FUNCTION "MOTOR" : VOID	// FC 101
AUTHOR : gaw-be
FAMILY : MOTOR
NAME : MOTOR
VERSION : 0.1
BEGIN
// (block stored without names or comments; labels and parameter names are numbered)
NETWORK
TITLE =
      BLD   5;
      T     LD 103;
      TAK;
      T     LD 107;
      L     P##PARAM9;
      LAR1;
      L     W [AR1,P#0.0];
      T     LW 101;
      OPN   DB [LW 101];
      L     D [AR1,P#2.0];
      LAR1;
      L     LD 107;
      L     LD 103;
      L     W [AR1,P#2.0];
      L     -1;
      ==I;
      BLD   5;
      T     LD 103;
      TAK;
      T     LD 107;
      L     P##PARAM9;
      LAR1;
      L     W [AR1,P#0.0];
      T     LW 101;
      OPN   DB [LW 101];
      L     D [AR1,P#2.0];
      LAR1;
      L     LD 107;
      L     LD 103;
      R      [AR1,P#4.0];
      L     #PARAM5;
      BLD   5;
      T     LD 103;
      TAK;
      T     LD 107;
      L     P##PARAM9;
      LAR1;
      L     W [AR1,P#0.0];
      T     LW 101;
      OPN   DB [LW 101];
      L     D [AR1,P#2.0];
      LAR1;
      L     LD 107;
      L     LD 103;
      L     W [AR1,P#2.0];
      <>I;
      JC    M002;
      BLD   5;
      T     LD 103;
      TAK;
      T     LD 107;
      L     P##PARAM9;
      LAR1;
      L     W [AR1,P#0.0];
      T     LW 101;
      OPN   DB [LW 101];
      L     D [AR1,P#2.0];
      LAR1;
      L     LD 107;
      L     LD 103;
      A      [AR1,P#4.0];
      JC    M001;
      BLD   5;
      T     LD 103;
      TAK;
      T     LD 107;
      L     P##PARAM8;
      LAR1;
      L     W [AR1,P#0.0];
      T     LW 101;
      OPN   DB [LW 101];
      L     D [AR1,P#2.0];
      LAR1;
      L     LD 107;
      L     LD 103;
      A      [AR1,P#0.0];
      BLD   5;
      T     LD 103;
      TAK;
      T     LD 107;
      L     P##PARAM9;
      LAR1;
      L     W [AR1,P#0.0];
      T     LW 101;
      OPN   DB [LW 101];
      L     D [AR1,P#2.0];
      LAR1;
      L     LD 107;
      L     LD 103;
      =      [AR1,P#0.0];
      BLD   5;
      T     LD 103;
      TAK;
      T     LD 107;
      L     P##PARAM8;
      LAR1;
      L     W [AR1,P#0.0];
      T     LW 101;
      OPN   DB [LW 101];
      L     D [AR1,P#2.0];
      LAR1;
      L     LD 107;
      L     LD 103;
      A      [AR1,P#0.1];
      BLD   5;
      T     LD 103;
      TAK;
      T     LD 107;
      L     P##PARAM9;
      LAR1;
      L     W [AR1,P#0.0];
      T     LW 101;
      OPN   DB [LW 101];
      L     D [AR1,P#2.0];
      LAR1;
      L     LD 107;
      L     LD 103;
      =      [AR1,P#0.1];
      BLD   5;
      T     LD 103;
      TAK;
      T     LD 107;
      L     P##PARAM8;
      LAR1;
      L     W [AR1,P#0.0];
      T     LW 101;
      OPN   DB [LW 101];
      L     D [AR1,P#2.0];
      LAR1;
      L     LD 107;
      L     LD 103;
      A      [AR1,P#0.3];
      BLD   5;
      T     LD 103;
      TAK;
      T     LD 107;
      L     P##PARAM9;
      LAR1;
      L     W [AR1,P#0.0];
      T     LW 101;
      OPN   DB [LW 101];
      L     D [AR1,P#2.0];
      LAR1;
      L     LD 107;
      L     LD 103;
      =      [AR1,P#0.3];
      SET;
      BLD   5;
      T     LD 103;
      TAK;
      T     LD 107;
      L     P##PARAM9;
      LAR1;
      L     W [AR1,P#0.0];
      T     LW 101;
      OPN   DB [LW 101];
      L     D [AR1,P#2.0];
      LAR1;
      L     LD 107;
      L     LD 103;
      =      [AR1,P#4.0];
M001: BLD   5;
      T     LD 103;
      TAK;
      T     LD 107;
      L     P##PARAM9;
      LAR1;
      L     W [AR1,P#0.0];
      T     LW 101;
      OPN   DB [LW 101];
      L     D [AR1,P#2.0];
      LAR1;
      L     LD 107;
      L     LD 103;
      A      [AR1,P#0.0];
      BLD   5;
      T     LD 103;
      TAK;
      T     LD 107;
      L     P##PARAM8;
      LAR1;
      L     W [AR1,P#0.0];
      T     LW 101;
      OPN   DB [LW 101];
      L     D [AR1,P#2.0];
      LAR1;
      L     LD 107;
      L     LD 103;
      =      [AR1,P#0.0];
      BLD   5;
      T     LD 103;
      TAK;
      T     LD 107;
      L     P##PARAM9;
      LAR1;
      L     W [AR1,P#0.0];
      T     LW 101;
      OPN   DB [LW 101];
      L     D [AR1,P#2.0];
      LAR1;
      L     LD 107;
      L     LD 103;
      A      [AR1,P#0.1];
      BLD   5;
      T     LD 103;
      TAK;
      T     LD 107;
      L     P##PARAM8;
      LAR1;
      L     W [AR1,P#0.0];
      T     LW 101;
      OPN   DB [LW 101];
      L     D [AR1,P#2.0];
      LAR1;
      L     LD 107;
      L     LD 103;
      =      [AR1,P#0.1];
      BLD   5;
      T     LD 103;
      TAK;
      T     LD 107;
      L     P##PARAM8;
      LAR1;
      L     W [AR1,P#0.0];
      T     LW 101;
      OPN   DB [LW 101];
      L     D [AR1,P#2.0];
      LAR1;
      L     LD 107;
      L     LD 103;
      A      [AR1,P#0.2];
      BLD   5;
      T     LD 103;
      TAK;
      T     LD 107;
      L     P##PARAM9;
      LAR1;
      L     W [AR1,P#0.0];
      T     LW 101;
      OPN   DB [LW 101];
      L     D [AR1,P#2.0];
      LAR1;
      L     LD 107;
      L     LD 103;
      =      [AR1,P#0.2];
      BLD   5;
      T     LD 103;
      TAK;
      T     LD 107;
      L     P##PARAM9;
      LAR1;
      L     W [AR1,P#0.0];
      T     LW 101;
      OPN   DB [LW 101];
      L     D [AR1,P#2.0];
      LAR1;
      L     LD 107;
      L     LD 103;
      A      [AR1,P#0.3];
      BLD   5;
      T     LD 103;
      TAK;
      T     LD 107;
      L     P##PARAM8;
      LAR1;
      L     W [AR1,P#0.0];
      T     LW 101;
      OPN   DB [LW 101];
      L     D [AR1,P#2.0];
      LAR1;
      L     LD 107;
      L     LD 103;
      =      [AR1,P#0.3];
      BLD   5;
      T     LD 103;
      TAK;
      T     LD 107;
      L     P##PARAM8;
      LAR1;
      L     W [AR1,P#0.0];
      T     LW 101;
      OPN   DB [LW 101];
      L     D [AR1,P#2.0];
      LAR1;
      L     LD 107;
      L     LD 103;
      A      [AR1,P#0.4];
      BLD   5;
      T     LD 103;
      TAK;
      T     LD 107;
      L     P##PARAM9;
      LAR1;
      L     W [AR1,P#0.0];
      T     LW 101;
      OPN   DB [LW 101];
      L     D [AR1,P#2.0];
      LAR1;
      L     LD 107;
      L     LD 103;
      =      [AR1,P#0.4];
      BLD   5;
      T     LD 103;
      TAK;
      T     LD 107;
      L     P##PARAM8;
      LAR1;
      L     W [AR1,P#0.0];
      T     LW 101;
      OPN   DB [LW 101];
      L     D [AR1,P#2.0];
      LAR1;
      L     LD 107;
      L     LD 103;
      A      [AR1,P#0.5];
      BLD   5;
      T     LD 103;
      TAK;
      T     LD 107;
      L     P##PARAM9;
      LAR1;
      L     W [AR1,P#0.0];
      T     LW 101;
      OPN   DB [LW 101];
      L     D [AR1,P#2.0];
      LAR1;
      L     LD 107;
      L     LD 103;
      =      [AR1,P#0.5];
      BLD   5;
      T     LD 103;
      TAK;
      T     LD 107;
      L     P##PARAM8;
      LAR1;
      L     W [AR1,P#0.0];
      T     LW 101;
      OPN   DB [LW 101];
      L     D [AR1,P#2.0];
      LAR1;
      L     LD 107;
      L     LD 103;
      A      [AR1,P#0.6];
      BLD   5;
      T     LD 103;
      TAK;
      T     LD 107;
      L     P##PARAM9;
      LAR1;
      L     W [AR1,P#0.0];
      T     LW 101;
      OPN   DB [LW 101];
      L     D [AR1,P#2.0];
      LAR1;
      L     LD 107;
      L     LD 103;
      =      [AR1,P#0.6];
      BLD   5;
      T     LD 103;
      TAK;
      T     LD 107;
      L     P##PARAM8;
      LAR1;
      L     W [AR1,P#0.0];
      T     LW 101;
      OPN   DB [LW 101];
      L     D [AR1,P#2.0];
      LAR1;
      L     LD 107;
      L     LD 103;
      A      [AR1,P#0.7];
      BLD   5;
      T     LD 103;
      TAK;
      T     LD 107;
      L     P##PARAM9;
      LAR1;
      L     W [AR1,P#0.0];
      T     LW 101;
      OPN   DB [LW 101];
      L     D [AR1,P#2.0];
      LAR1;
      L     LD 107;
      L     LD 103;
      =      [AR1,P#0.7];
      BLD   5;
      T     LD 103;
      TAK;
      T     LD 107;
      L     P##PARAM8;
      LAR1;
      L     W [AR1,P#0.0];
      T     LW 101;
      OPN   DB [LW 101];
      L     D [AR1,P#2.0];
      LAR1;
      L     LD 107;
      L     LD 103;
      L     B [AR1,P#1.0];
      BLD   5;
      T     LD 103;
      TAK;
      T     LD 107;
      L     P##PARAM9;
      LAR1;
      L     W [AR1,P#0.0];
      T     LW 101;
      OPN   DB [LW 101];
      L     D [AR1,P#2.0];
      LAR1;
      L     LD 107;
      L     LD 103;
      T     B [AR1,P#1.0];
M002: NOP   0;
NETWORK
TITLE =
      A(;
      A     #PARAM3;
      BLD   5;
      T     LD 103;
      TAK;
      T     LD 107;
      L     P##PARAM8;
      LAR1;
      L     W [AR1,P#0.0];
      T     LW 101;
      OPN   DB [LW 101];
      L     D [AR1,P#2.0];
      LAR1;
      L     LD 107;
      L     LD 103;
      AN     [AR1,P#0.0];
      O;
      BLD   5;
      T     LD 103;
      TAK;
      T     LD 107;
      L     P##PARAM8;
      LAR1;
      L     W [AR1,P#0.0];
      T     LW 101;
      OPN   DB [LW 101];
      L     D [AR1,P#2.0];
      LAR1;
      L     LD 107;
      L     LD 103;
      A      [AR1,P#0.0];
      BLD   5;
      T     LD 103;
      TAK;
      T     LD 107;
      L     P##PARAM8;
      LAR1;
      L     W [AR1,P#0.0];
      T     LW 101;
      OPN   DB [LW 101];
      L     D [AR1,P#2.0];
      LAR1;
      L     LD 107;
      L     LD 103;
      A      [AR1,P#0.1];
      );
      AN    #PARAM4;
      AN    #PARAM2;
      =     L 0.0;
      =     #PARAM6;
NETWORK
TITLE =
      A     #PARAM2;
      BLD   5;
      T     LD 103;
      TAK;
      T     LD 107;
      L     P##PARAM8;
      LAR1;
      L     W [AR1,P#0.0];
      T     LW 101;
      OPN   DB [LW 101];
      L     D [AR1,P#2.0];
      LAR1;
      L     LD 107;
      L     LD 103;
      =      [AR1,P#0.2];
NETWORK
TITLE =
      BLD   5;
      T     LD 103;
      TAK;
      T     LD 107;
      L     P##PARAM8;
      LAR1;
      L     W [AR1,P#0.0];
      T     LW 101;
      OPN   DB [LW 101];
      L     D [AR1,P#2.0];
      LAR1;
      L     LD 107;
      L     LD 103;
      A      [AR1,P#0.2];
      BLD   5;
      T     LD 103;
      TAK;
      T     LD 107;
      L     P##PARAM8;
      LAR1;
      L     W [AR1,P#0.0];
      T     LW 101;
      OPN   DB [LW 101];
      L     D [AR1,P#2.0];
      LAR1;
      L     LD 107;
      L     LD 103;
      A      [AR1,P#0.3];
      BLD   5;
      T     LD 103;
      TAK;
      T     LD 107;
      L     P##PARAM8;
      LAR1;
      L     W [AR1,P#0.0];
      T     LW 101;
      OPN   DB [LW 101];
      L     D [AR1,P#2.0];
      LAR1;
      L     LD 107;
      L     LD 103;
      R      [AR1,P#0.2];
NETWORK
TITLE =
      A     L 0.0;
      AN    #PARAM1;
      O;
      AN    L 0.0;
      A     #PARAM1;
      BLD   5;
      T     LD 103;
      TAK;
      T     LD 107;
      L     P##PARAM8;
      LAR1;
      L     W [AR1,P#0.0];
      T     LW 101;
      OPN   DB [LW 101];
      L     D [AR1,P#2.0];
      LAR1;
      L     LD 107;
      L     LD 103;
      O      [AR1,P#0.2];
      =     #PARAM7;
NETWORK
TITLE =
      AN    #PARAM1;
      AN    #PARAM2;
      BLD   5;
      T     LD 103;
      TAK;
      T     LD 107;
      L     P##PARAM8;
      LAR1;
      L     W [AR1,P#0.0];
      T     LW 101;
      OPN   DB [LW 101];
      L     D [AR1,P#2.0];
      LAR1;
      L     LD 107;
      L     LD 103;
      =      [AR1,P#0.4];
NETWORK
TITLE =
      A     #PARAM1;
      AN    #PARAM2;
      BLD   5;
      T     LD 103;
      TAK;
      T     LD 107;
      L     P##PARAM8;
      LAR1;
      L     W [AR1,P#0.0];
      T     LW 101;
      OPN   DB [LW 101];
      L     D [AR1,P#2.0];
      LAR1;
      L     LD 107;
      L     LD 103;
      =      [AR1,P#0.5];
NETWORK
TITLE =
      A     #PARAM2;
      A     M 0.7;
      BLD   5;
      T     LD 103;
      TAK;
      T     LD 107;
      L     P##PARAM8;
      LAR1;
      L     W [AR1,P#0.0];
      T     LW 101;
      OPN   DB [LW 101];
      L     D [AR1,P#2.0];
      LAR1;
      L     LD 107;
      L     LD 103;
      =      [AR1,P#0.6];
NETWORK
TITLE =
      A     #PARAM2;
      AN    M 0.7;
      BLD   5;
      T     LD 103;
      TAK;
      T     LD 107;
      L     P##PARAM8;
      LAR1;
      L     W [AR1,P#0.0];
      T     LW 101;
      OPN   DB [LW 101];
      L     D [AR1,P#2.0];
      LAR1;
      L     LD 107;
      L     LD 103;
      =      [AR1,P#0.7];
NETWORK
TITLE =
      BLD   5;
      T     LD 103;
      TAK;
      T     LD 107;
      L     P##PARAM8;
      LAR1;
      L     W [AR1,P#0.0];
      T     LW 101;
      OPN   DB [LW 101];
      L     D [AR1,P#2.0];
      LAR1;
      L     LD 107;
      L     LD 103;
      A      [AR1,P#0.3];
      BLD   5;
      T     LD 103;
      TAK;
      T     LD 107;
      L     P##PARAM8;
      LAR1;
      L     W [AR1,P#0.0];
      T     LW 101;
      OPN   DB [LW 101];
      L     D [AR1,P#2.0];
      LAR1;
      L     LD 107;
      L     LD 103;
      R      [AR1,P#0.3];
NETWORK
TITLE =
      BLD   5;
      T     LD 103;
      TAK;
      T     LD 107;
      L     P##PARAM8;
      LAR1;
      L     W [AR1,P#0.0];
      T     LW 101;
      OPN   DB [LW 101];
      L     D [AR1,P#2.0];
      LAR1;
      L     LD 107;
      L     LD 103;
      A      [AR1,P#0.0];
      =     L 100.0;
      BLD   5;
      T     LD 103;
      TAK;
      T     LD 107;
      L     P##PARAM8;
      LAR1;
      L     W [AR1,P#0.0];
      T     LW 101;
      OPN   DB [LW 101];
      L     D [AR1,P#2.0];
      LAR1;
      L     LD 107;
      L     LD 103;
      A      [AR1,P#0.1];
      =     L 100.1;
      BLD   5;
      T     LD 103;
      TAK;
      T     LD 107;
      L     P##PARAM8;
      LAR1;
      L     W [AR1,P#0.0];
      T     LW 101;
      OPN   DB [LW 101];
      L     D [AR1,P#2.0];
      LAR1;
      L     LD 107;
      L     LD 103;
      A      [AR1,P#0.2];
      =     L 100.2;
      BLD   5;
      T     LD 103;
      TAK;
      T     LD 107;
      L     P##PARAM8;
      LAR1;
      L     W [AR1,P#0.0];
      T     LW 101;
      OPN   DB [LW 101];
      L     D [AR1,P#2.0];
      LAR1;
      L     LD 107;
      L     LD 103;
      A      [AR1,P#0.3];
      =     L 100.3;
      BLD   5;
      T     LD 103;
      TAK;
      T     LD 107;
      L     P##PARAM8;
      LAR1;
      L     W [AR1,P#0.0];
      T     LW 101;
      OPN   DB [LW 101];
      L     D [AR1,P#2.0];
      LAR1;
      L     LD 107;
      L     LD 103;
      A      [AR1,P#0.4];
      =     L 100.4;
      BLD   5;
      T     LD 103;
      TAK;
      T     LD 107;
      L     P##PARAM8;
      LAR1;
      L     W [AR1,P#0.0];
      T     LW 101;
      OPN   DB [LW 101];
      L     D [AR1,P#2.0];
      LAR1;
      L     LD 107;
      L     LD 103;
      A      [AR1,P#0.5];
      =     L 100.5;
      BLD   5;
      T     LD 103;
      TAK;
      T     LD 107;
      L     P##PARAM8;
      LAR1;
      L     W [AR1,P#0.0];
      T     LW 101;
      OPN   DB [LW 101];
      L     D [AR1,P#2.0];
      LAR1;
      L     LD 107;
      L     LD 103;
      A      [AR1,P#0.6];
      =     L 100.6;
      BLD   5;
      T     LD 103;
      TAK;
      T     LD 107;
      L     P##PARAM8;
      LAR1;
      L     W [AR1,P#0.0];
      T     LW 101;
      OPN   DB [LW 101];
      L     D [AR1,P#2.0];
      LAR1;
      L     LD 107;
      L     LD 103;
      A      [AR1,P#0.7];
      =     L 100.7;
      L     LB 100;
      BLD   5;
      T     LD 103;
      TAK;
      T     LD 107;
      L     P##PARAM8;
      LAR1;
      L     W [AR1,P#0.0];
      T     LW 101;
      OPN   DB [LW 101];
      L     D [AR1,P#2.0];
      LAR1;
      L     LD 107;
      L     LD 103;
      T     B [AR1,P#1.0];
END_FUNCTION

FUNCTION "level" : VOID	// FC 107
AUTHOR : gaw-be
FAMILY : level
NAME : display
VERSION : 0.2
BEGIN
// (block stored without names or comments; labels and parameter names are numbered)
NETWORK
TITLE =
      L     #PARAM3;
      BLD   5;
      T     LD 106;
      TAK;
      T     LD 110;
      L     P##PARAM12;
      LAR1;
      L     W [AR1,P#0.0];
      T     LW 104;
      OPN   DB [LW 104];
      L     D [AR1,P#2.0];
      LAR1;
      L     LD 110;
      L     LD 106;
      T     B [AR1,P#28.0];
      BLD   5;
      T     LD 106;
      TAK;
      T     LD 110;
      L     P##PARAM13;
      LAR1;
      L     W [AR1,P#0.0];
      T     LW 104;
      OPN   DB [LW 104];
      L     D [AR1,P#2.0];
      LAR1;
      L     LD 110;
      L     LD 106;
      L     W [AR1,P#28.0];
      L     -1;
      ==I;
      BLD   5;
      T     LD 106;
      TAK;
      T     LD 110;
      L     P##PARAM13;
      LAR1;
      L     W [AR1,P#0.0];
      T     LW 104;
      OPN   DB [LW 104];
      L     D [AR1,P#2.0];
      LAR1;
      L     LD 110;
      L     LD 106;
      R      [AR1,P#30.0];
      L     #PARAM2;
      BLD   5;
      T     LD 106;
      TAK;
      T     LD 110;
      L     P##PARAM13;
      LAR1;
      L     W [AR1,P#0.0];
      T     LW 104;
      OPN   DB [LW 104];
      L     D [AR1,P#2.0];
      LAR1;
      L     LD 110;
      L     LD 106;
      L     W [AR1,P#28.0];
      <>I;
      JC    M010;
      BLD   5;
      T     LD 106;
      TAK;
      T     LD 110;
      L     P##PARAM13;
      LAR1;
      L     W [AR1,P#0.0];
      T     LW 104;
      OPN   DB [LW 104];
      L     D [AR1,P#2.0];
      LAR1;
      L     LD 110;
      L     LD 106;
      A      [AR1,P#30.0];
      JC    M001;
      BLD   5;
      T     LD 106;
      TAK;
      T     LD 110;
      L     P##PARAM12;
      LAR1;
      L     W [AR1,P#0.0];
      T     LW 104;
      OPN   DB [LW 104];
      L     D [AR1,P#2.0];
      LAR1;
      L     LD 110;
      L     LD 106;
      L     B [AR1,P#4.0];
      BLD   5;
      T     LD 106;
      TAK;
      T     LD 110;
      L     P##PARAM13;
      LAR1;
      L     W [AR1,P#0.0];
      T     LW 104;
      OPN   DB [LW 104];
      L     D [AR1,P#2.0];
      LAR1;
      L     LD 110;
      L     LD 106;
      T     B [AR1,P#4.0];
      BLD   5;
      T     LD 106;
      TAK;
      T     LD 110;
      L     P##PARAM12;
      LAR1;
      L     W [AR1,P#0.0];
      T     LW 104;
      OPN   DB [LW 104];
      L     D [AR1,P#2.0];
      LAR1;
      L     LD 110;
      L     LD 106;
      L     D [AR1,P#6.0];
      BLD   5;
      T     LD 106;
      TAK;
      T     LD 110;
      L     P##PARAM13;
      LAR1;
      L     W [AR1,P#0.0];
      T     LW 104;
      OPN   DB [LW 104];
      L     D [AR1,P#2.0];
      LAR1;
      L     LD 110;
      L     LD 106;
      T     D [AR1,P#6.0];
      BLD   5;
      T     LD 106;
      TAK;
      T     LD 110;
      L     P##PARAM12;
      LAR1;
      L     W [AR1,P#0.0];
      T     LW 104;
      OPN   DB [LW 104];
      L     D [AR1,P#2.0];
      LAR1;
      L     LD 110;
      L     LD 106;
      L     D [AR1,P#10.0];
      BLD   5;
      T     LD 106;
      TAK;
      T     LD 110;
      L     P##PARAM13;
      LAR1;
      L     W [AR1,P#0.0];
      T     LW 104;
      OPN   DB [LW 104];
      L     D [AR1,P#2.0];
      LAR1;
      L     LD 110;
      L     LD 106;
      T     D [AR1,P#10.0];
      BLD   5;
      T     LD 106;
      TAK;
      T     LD 110;
      L     P##PARAM12;
      LAR1;
      L     W [AR1,P#0.0];
      T     LW 104;
      OPN   DB [LW 104];
      L     D [AR1,P#2.0];
      LAR1;
      L     LD 110;
      L     LD 106;
      L     D [AR1,P#14.0];
      BLD   5;
      T     LD 106;
      TAK;
      T     LD 110;
      L     P##PARAM13;
      LAR1;
      L     W [AR1,P#0.0];
      T     LW 104;
      OPN   DB [LW 104];
      L     D [AR1,P#2.0];
      LAR1;
      L     LD 110;
      L     LD 106;
      T     D [AR1,P#14.0];
      BLD   5;
      T     LD 106;
      TAK;
      T     LD 110;
      L     P##PARAM12;
      LAR1;
      L     W [AR1,P#0.0];
      T     LW 104;
      OPN   DB [LW 104];
      L     D [AR1,P#2.0];
      LAR1;
      L     LD 110;
      L     LD 106;
      L     W [AR1,P#18.0];
      BLD   5;
      T     LD 106;
      TAK;
      T     LD 110;
      L     P##PARAM13;
      LAR1;
      L     W [AR1,P#0.0];
      T     LW 104;
      OPN   DB [LW 104];
      L     D [AR1,P#2.0];
      LAR1;
      L     LD 110;
      L     LD 106;
      T     W [AR1,P#18.0];
      BLD   5;
      T     LD 106;
      TAK;
      T     LD 110;
      L     P##PARAM12;
      LAR1;
      L     W [AR1,P#0.0];
      T     LW 104;
      OPN   DB [LW 104];
      L     D [AR1,P#2.0];
      LAR1;
      L     LD 110;
      L     LD 106;
      L     W [AR1,P#20.0];
      BLD   5;
      T     LD 106;
      TAK;
      T     LD 110;
      L     P##PARAM13;
      LAR1;
      L     W [AR1,P#0.0];
      T     LW 104;
      OPN   DB [LW 104];
      L     D [AR1,P#2.0];
      LAR1;
      L     LD 110;
      L     LD 106;
      T     W [AR1,P#20.0];
      BLD   5;
      T     LD 106;
      TAK;
      T     LD 110;
      L     P##PARAM12;
      LAR1;
      L     W [AR1,P#0.0];
      T     LW 104;
      OPN   DB [LW 104];
      L     D [AR1,P#2.0];
      LAR1;
      L     LD 110;
      L     LD 106;
      L     W [AR1,P#22.0];
      BLD   5;
      T     LD 106;
      TAK;
      T     LD 110;
      L     P##PARAM13;
      LAR1;
      L     W [AR1,P#0.0];
      T     LW 104;
      OPN   DB [LW 104];
      L     D [AR1,P#2.0];
      LAR1;
      L     LD 110;
      L     LD 106;
      T     W [AR1,P#22.0];
      BLD   5;
      T     LD 106;
      TAK;
      T     LD 110;
      L     P##PARAM12;
      LAR1;
      L     W [AR1,P#0.0];
      T     LW 104;
      OPN   DB [LW 104];
      L     D [AR1,P#2.0];
      LAR1;
      L     LD 110;
      L     LD 106;
      L     W [AR1,P#24.0];
      BLD   5;
      T     LD 106;
      TAK;
      T     LD 110;
      L     P##PARAM13;
      LAR1;
      L     W [AR1,P#0.0];
      T     LW 104;
      OPN   DB [LW 104];
      L     D [AR1,P#2.0];
      LAR1;
      L     LD 110;
      L     LD 106;
      T     W [AR1,P#24.0];
      BLD   5;
      T     LD 106;
      TAK;
      T     LD 110;
      L     P##PARAM12;
      LAR1;
      L     W [AR1,P#0.0];
      T     LW 104;
      OPN   DB [LW 104];
      L     D [AR1,P#2.0];
      LAR1;
      L     LD 110;
      L     LD 106;
      L     W [AR1,P#26.0];
      BLD   5;
      T     LD 106;
      TAK;
      T     LD 110;
      L     P##PARAM13;
      LAR1;
      L     W [AR1,P#0.0];
      T     LW 104;
      OPN   DB [LW 104];
      L     D [AR1,P#2.0];
      LAR1;
      L     LD 110;
      L     LD 106;
      T     W [AR1,P#26.0];
      BLD   5;
      T     LD 106;
      TAK;
      T     LD 110;
      L     P##PARAM12;
      LAR1;
      L     W [AR1,P#0.0];
      T     LW 104;
      OPN   DB [LW 104];
      L     D [AR1,P#2.0];
      LAR1;
      L     LD 110;
      L     LD 106;
      L     B [AR1,P#28.0];
      BLD   5;
      T     LD 106;
      TAK;
      T     LD 110;
      L     P##PARAM13;
      LAR1;
      L     W [AR1,P#0.0];
      T     LW 104;
      OPN   DB [LW 104];
      L     D [AR1,P#2.0];
      LAR1;
      L     LD 110;
      L     LD 106;
      T     B [AR1,P#31.0];
      BLD   5;
      T     LD 106;
      TAK;
      T     LD 110;
      L     P##PARAM12;
      LAR1;
      L     W [AR1,P#0.0];
      T     LW 104;
      OPN   DB [LW 104];
      L     D [AR1,P#2.0];
      LAR1;
      L     LD 110;
      L     LD 106;
      L     W [AR1,P#30.0];
      BLD   5;
      T     LD 106;
      TAK;
      T     LD 110;
      L     P##PARAM13;
      LAR1;
      L     W [AR1,P#0.0];
      T     LW 104;
      OPN   DB [LW 104];
      L     D [AR1,P#2.0];
      LAR1;
      L     LD 110;
      L     LD 106;
      T     W [AR1,P#32.0];
      BLD   5;
      T     LD 106;
      TAK;
      T     LD 110;
      L     P##PARAM12;
      LAR1;
      L     W [AR1,P#0.0];
      T     LW 104;
      OPN   DB [LW 104];
      L     D [AR1,P#2.0];
      LAR1;
      L     LD 110;
      L     LD 106;
      L     W [AR1,P#32.0];
      BLD   5;
      T     LD 106;
      TAK;
      T     LD 110;
      L     P##PARAM13;
      LAR1;
      L     W [AR1,P#0.0];
      T     LW 104;
      OPN   DB [LW 104];
      L     D [AR1,P#2.0];
      LAR1;
      L     LD 110;
      L     LD 106;
      T     W [AR1,P#34.0];
      BLD   5;
      T     LD 106;
      TAK;
      T     LD 110;
      L     P##PARAM12;
      LAR1;
      L     W [AR1,P#0.0];
      T     LW 104;
      OPN   DB [LW 104];
      L     D [AR1,P#2.0];
      LAR1;
      L     LD 110;
      L     LD 106;
      L     W [AR1,P#34.0];
      BLD   5;
      T     LD 106;
      TAK;
      T     LD 110;
      L     P##PARAM13;
      LAR1;
      L     W [AR1,P#0.0];
      T     LW 104;
      OPN   DB [LW 104];
      L     D [AR1,P#2.0];
      LAR1;
      L     LD 110;
      L     LD 106;
      T     W [AR1,P#36.0];
      BLD   5;
      T     LD 106;
      TAK;
      T     LD 110;
      L     P##PARAM12;
      LAR1;
      L     W [AR1,P#0.0];
      T     LW 104;
      OPN   DB [LW 104];
      L     D [AR1,P#2.0];
      LAR1;
      L     LD 110;
      L     LD 106;
      L     W [AR1,P#36.0];
      BLD   5;
      T     LD 106;
      TAK;
      T     LD 110;
      L     P##PARAM13;
      LAR1;
      L     W [AR1,P#0.0];
      T     LW 104;
      OPN   DB [LW 104];
      L     D [AR1,P#2.0];
      LAR1;
      L     LD 110;
      L     LD 106;
      T     W [AR1,P#38.0];
      BLD   5;
      T     LD 106;
      TAK;
      T     LD 110;
      L     P##PARAM12;
      LAR1;
      L     W [AR1,P#0.0];
      T     LW 104;
      OPN   DB [LW 104];
      L     D [AR1,P#2.0];
      LAR1;
      L     LD 110;
      L     LD 106;
      L     W [AR1,P#38.0];
      BLD   5;
      T     LD 106;
      TAK;
      T     LD 110;
      L     P##PARAM13;
      LAR1;
      L     W [AR1,P#0.0];
      T     LW 104;
      OPN   DB [LW 104];
      L     D [AR1,P#2.0];
      LAR1;
      L     LD 110;
      L     LD 106;
      T     W [AR1,P#40.0];
      BLD   5;
      T     LD 106;
      TAK;
      T     LD 110;
      L     P##PARAM12;
      LAR1;
      L     W [AR1,P#0.0];
      T     LW 104;
      OPN   DB [LW 104];
      L     D [AR1,P#2.0];
      LAR1;
      L     LD 110;
      L     LD 106;
      L     W [AR1,P#40.0];
      BLD   5;
      T     LD 106;
      TAK;
      T     LD 110;
      L     P##PARAM13;
      LAR1;
      L     W [AR1,P#0.0];
      T     LW 104;
      OPN   DB [LW 104];
      L     D [AR1,P#2.0];
      LAR1;
      L     LD 110;
      L     LD 106;
      T     W [AR1,P#42.0];
      BLD   5;
      T     LD 106;
      TAK;
      T     LD 110;
      L     P##PARAM12;
      LAR1;
      L     W [AR1,P#0.0];
      T     LW 104;
      OPN   DB [LW 104];
      L     D [AR1,P#2.0];
      LAR1;
      L     LD 110;
      L     LD 106;
      L     W [AR1,P#42.0];
      BLD   5;
      T     LD 106;
      TAK;
      T     LD 110;
      L     P##PARAM13;
      LAR1;
      L     W [AR1,P#0.0];
      T     LW 104;
      OPN   DB [LW 104];
      L     D [AR1,P#2.0];
      LAR1;
      L     LD 110;
      L     LD 106;
      T     W [AR1,P#44.0];
      BLD   5;
      T     LD 106;
      TAK;
      T     LD 110;
      L     P##PARAM12;
      LAR1;
      L     W [AR1,P#0.0];
      T     LW 104;
      OPN   DB [LW 104];
      L     D [AR1,P#2.0];
      LAR1;
      L     LD 110;
      L     LD 106;
      L     W [AR1,P#44.0];
      BLD   5;
      T     LD 106;
      TAK;
      T     LD 110;
      L     P##PARAM13;
      LAR1;
      L     W [AR1,P#0.0];
      T     LW 104;
      OPN   DB [LW 104];
      L     D [AR1,P#2.0];
      LAR1;
      L     LD 110;
      L     LD 106;
      T     W [AR1,P#46.0];
      SET;
      BLD   5;
      T     LD 106;
      TAK;
      T     LD 110;
      L     P##PARAM13;
      LAR1;
      L     W [AR1,P#0.0];
      T     LW 104;
      OPN   DB [LW 104];
      L     D [AR1,P#2.0];
      LAR1;
      L     LD 110;
      L     LD 106;
      =      [AR1,P#30.0];
M001: BLD   5;
      T     LD 106;
      TAK;
      T     LD 110;
      L     P##PARAM12;
      LAR1;
      L     W [AR1,P#0.0];
      T     LW 104;
      OPN   DB [LW 104];
      L     D [AR1,P#2.0];
      LAR1;
      L     LD 110;
      L     LD 106;
      L     D [AR1,P#0.0];
      BLD   5;
      T     LD 106;
      TAK;
      T     LD 110;
      L     P##PARAM13;
      LAR1;
      L     W [AR1,P#0.0];
      T     LW 104;
      OPN   DB [LW 104];
      L     D [AR1,P#2.0];
      LAR1;
      L     LD 110;
      L     LD 106;
      T     D [AR1,P#0.0];
      BLD   5;
      T     LD 106;
      TAK;
      T     LD 110;
      L     P##PARAM13;
      LAR1;
      L     W [AR1,P#0.0];
      T     LW 104;
      OPN   DB [LW 104];
      L     D [AR1,P#2.0];
      LAR1;
      L     LD 110;
      L     LD 106;
      L     B [AR1,P#4.0];
      BLD   5;
      T     LD 106;
      TAK;
      T     LD 110;
      L     P##PARAM12;
      LAR1;
      L     W [AR1,P#0.0];
      T     LW 104;
      OPN   DB [LW 104];
      L     D [AR1,P#2.0];
      LAR1;
      L     LD 110;
      L     LD 106;
      T     B [AR1,P#4.0];
      BLD   5;
      T     LD 106;
      TAK;
      T     LD 110;
      L     P##PARAM13;
      LAR1;
      L     W [AR1,P#0.0];
      T     LW 104;
      OPN   DB [LW 104];
      L     D [AR1,P#2.0];
      LAR1;
      L     LD 110;
      L     LD 106;
      L     D [AR1,P#10.0];
      BLD   5;
      T     LD 106;
      TAK;
      T     LD 110;
      L     P##PARAM12;
      LAR1;
      L     W [AR1,P#0.0];
      T     LW 104;
      OPN   DB [LW 104];
      L     D [AR1,P#2.0];
      LAR1;
      L     LD 110;
      L     LD 106;
      T     D [AR1,P#10.0];
      BLD   5;
      T     LD 106;
      TAK;
      T     LD 110;
      L     P##PARAM13;
      LAR1;
      L     W [AR1,P#0.0];
      T     LW 104;
      OPN   DB [LW 104];
      L     D [AR1,P#2.0];
      LAR1;
      L     LD 110;
      L     LD 106;
      L     D [AR1,P#14.0];
      L     3.000000e+00;
      >R;
      JC    M002;
      BLD   5;
      T     LD 106;
      TAK;
      T     LD 110;
      L     P##PARAM13;
      LAR1;
      L     W [AR1,P#0.0];
      T     LW 104;
      OPN   DB [LW 104];
      L     D [AR1,P#2.0];
      LAR1;
      L     LD 110;
      L     LD 106;
      L     D [AR1,P#14.0];
      L     8.000000e-01;
      <R;
      JC    M002;
      BLD   5;
      T     LD 106;
      TAK;
      T     LD 110;
      L     P##PARAM13;
      LAR1;
      L     W [AR1,P#0.0];
      T     LW 104;
      OPN   DB [LW 104];
      L     D [AR1,P#2.0];
      LAR1;
      L     LD 110;
      L     LD 106;
      L     D [AR1,P#14.0];
M002: BLD   5;
      T     LD 106;
      TAK;
      T     LD 110;
      L     P##PARAM13;
      LAR1;
      L     W [AR1,P#0.0];
      T     LW 104;
      OPN   DB [LW 104];
      L     D [AR1,P#2.0];
      LAR1;
      L     LD 110;
      L     LD 106;
      T     D [AR1,P#14.0];
      BLD   5;
      T     LD 106;
      TAK;
      T     LD 110;
      L     P##PARAM13;
      LAR1;
      L     W [AR1,P#0.0];
      T     LW 104;
      OPN   DB [LW 104];
      L     D [AR1,P#2.0];
      LAR1;
      L     LD 110;
      L     LD 106;
      L     D [AR1,P#14.0];
      BLD   5;
      T     LD 106;
      TAK;
      T     LD 110;
      L     P##PARAM12;
      LAR1;
      L     W [AR1,P#0.0];
      T     LW 104;
      OPN   DB [LW 104];
      L     D [AR1,P#2.0];
      LAR1;
      L     LD 110;
      L     LD 106;
      T     D [AR1,P#14.0];
      BLD   5;
      T     LD 106;
      TAK;
      T     LD 110;
      L     P##PARAM13;
      LAR1;
      L     W [AR1,P#0.0];
      T     LW 104;
      OPN   DB [LW 104];
      L     D [AR1,P#2.0];
      LAR1;
      L     LD 110;
      L     LD 106;
      L     D [AR1,P#6.0];
      BLD   5;
      T     LD 106;
      TAK;
      T     LD 110;
      L     P##PARAM13;
      LAR1;
      L     W [AR1,P#0.0];
      T     LW 104;
      OPN   DB [LW 104];
      L     D [AR1,P#2.0];
      LAR1;
      L     LD 110;
      L     LD 106;
      L     D [AR1,P#14.0];
      >R;
      JC    M003;
      BLD   5;
      T     LD 106;
      TAK;
      T     LD 110;
      L     P##PARAM13;
      LAR1;
      L     W [AR1,P#0.0];
      T     LW 104;
      OPN   DB [LW 104];
      L     D [AR1,P#2.0];
      LAR1;
      L     LD 110;
      L     LD 106;
      L     D [AR1,P#6.0];
      L     8.000000e-01;
      <R;
      JC    M003;
      BLD   5;
      T     LD 106;
      TAK;
      T     LD 110;
      L     P##PARAM13;
      LAR1;
      L     W [AR1,P#0.0];
      T     LW 104;
      OPN   DB [LW 104];
      L     D [AR1,P#2.0];
      LAR1;
      L     LD 110;
      L     LD 106;
      L     D [AR1,P#6.0];
M003: BLD   5;
      T     LD 106;
      TAK;
      T     LD 110;
      L     P##PARAM13;
      LAR1;
      L     W [AR1,P#0.0];
      T     LW 104;
      OPN   DB [LW 104];
      L     D [AR1,P#2.0];
      LAR1;
      L     LD 110;
      L     LD 106;
      T     D [AR1,P#6.0];
      BLD   5;
      T     LD 106;
      TAK;
      T     LD 110;
      L     P##PARAM13;
      LAR1;
      L     W [AR1,P#0.0];
      T     LW 104;
      OPN   DB [LW 104];
      L     D [AR1,P#2.0];
      LAR1;
      L     LD 110;
      L     LD 106;
      L     D [AR1,P#6.0];
      BLD   5;
      T     LD 106;
      TAK;
      T     LD 110;
      L     P##PARAM12;
      LAR1;
      L     W [AR1,P#0.0];
      T     LW 104;
      OPN   DB [LW 104];
      L     D [AR1,P#2.0];
      LAR1;
      L     LD 110;
      L     LD 106;
      T     D [AR1,P#6.0];
      BLD   5;
      T     LD 106;
      TAK;
      T     LD 110;
      L     P##PARAM13;
      LAR1;
      L     W [AR1,P#0.0];
      T     LW 104;
      OPN   DB [LW 104];
      L     D [AR1,P#2.0];
      LAR1;
      L     LD 110;
      L     LD 106;
      L     W [AR1,P#18.0];
      BLD   5;
      T     LD 106;
      TAK;
      T     LD 110;
      L     P##PARAM12;
      LAR1;
      L     W [AR1,P#0.0];
      T     LW 104;
      OPN   DB [LW 104];
      L     D [AR1,P#2.0];
      LAR1;
      L     LD 110;
      L     LD 106;
      T     W [AR1,P#18.0];
      BLD   5;
      T     LD 106;
      TAK;
      T     LD 110;
      L     P##PARAM13;
      LAR1;
      L     W [AR1,P#0.0];
      T     LW 104;
      OPN   DB [LW 104];
      L     D [AR1,P#2.0];
      LAR1;
      L     LD 110;
      L     LD 106;
      L     W [AR1,P#24.0];
      BLD   5;
      T     LD 106;
      TAK;
      T     LD 110;
      L     P##PARAM13;
      LAR1;
      L     W [AR1,P#0.0];
      T     LW 104;
      OPN   DB [LW 104];
      L     D [AR1,P#2.0];
      LAR1;
      L     LD 110;
      L     LD 106;
      L     W [AR1,P#26.0];
      >R;
      JC    M004;
      BLD   5;
      T     LD 106;
      TAK;
      T     LD 110;
      L     P##PARAM13;
      LAR1;
      L     W [AR1,P#0.0];
      T     LW 104;
      OPN   DB [LW 104];
      L     D [AR1,P#2.0];
      LAR1;
      L     LD 110;
      L     LD 106;
      L     W [AR1,P#24.0];
      BLD   5;
      T     LD 106;
      TAK;
      T     LD 110;
      L     P##PARAM13;
      LAR1;
      L     W [AR1,P#0.0];
      T     LW 104;
      OPN   DB [LW 104];
      L     D [AR1,P#2.0];
      LAR1;
      L     LD 110;
      L     LD 106;
      L     W [AR1,P#22.0];
      <R;
      JC    M004;
      BLD   5;
      T     LD 106;
      TAK;
      T     LD 110;
      L     P##PARAM13;
      LAR1;
      L     W [AR1,P#0.0];
      T     LW 104;
      OPN   DB [LW 104];
      L     D [AR1,P#2.0];
      LAR1;
      L     LD 110;
      L     LD 106;
      L     W [AR1,P#24.0];
M004: BLD   5;
      T     LD 106;
      TAK;
      T     LD 110;
      L     P##PARAM13;
      LAR1;
      L     W [AR1,P#0.0];
      T     LW 104;
      OPN   DB [LW 104];
      L     D [AR1,P#2.0];
      LAR1;
      L     LD 110;
      L     LD 106;
      T     W [AR1,P#24.0];
      BLD   5;
      T     LD 106;
      TAK;
      T     LD 110;
      L     P##PARAM13;
      LAR1;
      L     W [AR1,P#0.0];
      T     LW 104;
      OPN   DB [LW 104];
      L     D [AR1,P#2.0];
      LAR1;
      L     LD 110;
      L     LD 106;
      L     W [AR1,P#24.0];
      BLD   5;
      T     LD 106;
      TAK;
      T     LD 110;
      L     P##PARAM12;
      LAR1;
      L     W [AR1,P#0.0];
      T     LW 104;
      OPN   DB [LW 104];
      L     D [AR1,P#2.0];
      LAR1;
      L     LD 110;
      L     LD 106;
      T     W [AR1,P#24.0];
      BLD   5;
      T     LD 106;
      TAK;
      T     LD 110;
      L     P##PARAM13;
      LAR1;
      L     W [AR1,P#0.0];
      T     LW 104;
      OPN   DB [LW 104];
      L     D [AR1,P#2.0];
      LAR1;
      L     LD 110;
      L     LD 106;
      L     W [AR1,P#26.0];
      L     1.000000e+02;
      >R;
      JC    M005;
      BLD   5;
      T     LD 106;
      TAK;
      T     LD 110;
      L     P##PARAM13;
      LAR1;
      L     W [AR1,P#0.0];
      T     LW 104;
      OPN   DB [LW 104];
      L     D [AR1,P#2.0];
      LAR1;
      L     LD 110;
      L     LD 106;
      L     W [AR1,P#26.0];
      BLD   5;
      T     LD 106;
      TAK;
      T     LD 110;
      L     P##PARAM13;
      LAR1;
      L     W [AR1,P#0.0];
      T     LW 104;
      OPN   DB [LW 104];
      L     D [AR1,P#2.0];
      LAR1;
      L     LD 110;
      L     LD 106;
      L     W [AR1,P#24.0];
      <R;
      JC    M005;
      BLD   5;
      T     LD 106;
      TAK;
      T     LD 110;
      L     P##PARAM13;
      LAR1;
      L     W [AR1,P#0.0];
      T     LW 104;
      OPN   DB [LW 104];
      L     D [AR1,P#2.0];
      LAR1;
      L     LD 110;
      L     LD 106;
      L     W [AR1,P#26.0];
M005: BLD   5;
      T     LD 106;
      TAK;
      T     LD 110;
      L     P##PARAM13;
      LAR1;
      L     W [AR1,P#0.0];
      T     LW 104;
      OPN   DB [LW 104];
      L     D [AR1,P#2.0];
      LAR1;
      L     LD 110;
      L     LD 106;
      T     W [AR1,P#26.0];
      BLD   5;
      T     LD 106;
      TAK;
      T     LD 110;
      L     P##PARAM13;
      LAR1;
      L     W [AR1,P#0.0];
      T     LW 104;
      OPN   DB [LW 104];
      L     D [AR1,P#2.0];
      LAR1;
      L     LD 110;
      L     LD 106;
      L     W [AR1,P#26.0];
      BLD   5;
      T     LD 106;
      TAK;
      T     LD 110;
      L     P##PARAM12;
      LAR1;
      L     W [AR1,P#0.0];
      T     LW 104;
      OPN   DB [LW 104];
      L     D [AR1,P#2.0];
      LAR1;
      L     LD 110;
      L     LD 106;
      T     W [AR1,P#26.0];
      BLD   5;
      T     LD 106;
      TAK;
      T     LD 110;
      L     P##PARAM13;
      LAR1;
      L     W [AR1,P#0.0];
      T     LW 104;
      OPN   DB [LW 104];
      L     D [AR1,P#2.0];
      LAR1;
      L     LD 110;
      L     LD 106;
      L     W [AR1,P#22.0];
      BLD   5;
      T     LD 106;
      TAK;
      T     LD 110;
      L     P##PARAM13;
      LAR1;
      L     W [AR1,P#0.0];
      T     LW 104;
      OPN   DB [LW 104];
      L     D [AR1,P#2.0];
      LAR1;
      L     LD 110;
      L     LD 106;
      L     W [AR1,P#24.0];
      >R;
      JC    M006;
      BLD   5;
      T     LD 106;
      TAK;
      T     LD 110;
      L     P##PARAM13;
      LAR1;
      L     W [AR1,P#0.0];
      T     LW 104;
      OPN   DB [LW 104];
      L     D [AR1,P#2.0];
      LAR1;
      L     LD 110;
      L     LD 106;
      L     W [AR1,P#22.0];
      BLD   5;
      T     LD 106;
      TAK;
      T     LD 110;
      L     P##PARAM13;
      LAR1;
      L     W [AR1,P#0.0];
      T     LW 104;
      OPN   DB [LW 104];
      L     D [AR1,P#2.0];
      LAR1;
      L     LD 110;
      L     LD 106;
      L     W [AR1,P#20.0];
      <R;
      JC    M006;
      BLD   5;
      T     LD 106;
      TAK;
      T     LD 110;
      L     P##PARAM13;
      LAR1;
      L     W [AR1,P#0.0];
      T     LW 104;
      OPN   DB [LW 104];
      L     D [AR1,P#2.0];
      LAR1;
      L     LD 110;
      L     LD 106;
      L     W [AR1,P#22.0];
M006: BLD   5;
      T     LD 106;
      TAK;
      T     LD 110;
      L     P##PARAM13;
      LAR1;
      L     W [AR1,P#0.0];
      T     LW 104;
      OPN   DB [LW 104];
      L     D [AR1,P#2.0];
      LAR1;
      L     LD 110;
      L     LD 106;
      T     W [AR1,P#22.0];
      BLD   5;
      T     LD 106;
      TAK;
      T     LD 110;
      L     P##PARAM13;
      LAR1;
      L     W [AR1,P#0.0];
      T     LW 104;
      OPN   DB [LW 104];
      L     D [AR1,P#2.0];
      LAR1;
      L     LD 110;
      L     LD 106;
      L     W [AR1,P#22.0];
      BLD   5;
      T     LD 106;
      TAK;
      T     LD 110;
      L     P##PARAM12;
      LAR1;
      L     W [AR1,P#0.0];
      T     LW 104;
      OPN   DB [LW 104];
      L     D [AR1,P#2.0];
      LAR1;
      L     LD 110;
      L     LD 106;
      T     W [AR1,P#22.0];
      BLD   5;
      T     LD 106;
      TAK;
      T     LD 110;
      L     P##PARAM13;
      LAR1;
      L     W [AR1,P#0.0];
      T     LW 104;
      OPN   DB [LW 104];
      L     D [AR1,P#2.0];
      LAR1;
      L     LD 110;
      L     LD 106;
      L     W [AR1,P#20.0];
      BLD   5;
      T     LD 106;
      TAK;
      T     LD 110;
      L     P##PARAM13;
      LAR1;
      L     W [AR1,P#0.0];
      T     LW 104;
      OPN   DB [LW 104];
      L     D [AR1,P#2.0];
      LAR1;
      L     LD 110;
      L     LD 106;
      L     W [AR1,P#22.0];
      >R;
      JC    M007;
      BLD   5;
      T     LD 106;
      TAK;
      T     LD 110;
      L     P##PARAM13;
      LAR1;
      L     W [AR1,P#0.0];
      T     LW 104;
      OPN   DB [LW 104];
      L     D [AR1,P#2.0];
      LAR1;
      L     LD 110;
      L     LD 106;
      L     W [AR1,P#20.0];
      L     0.000000e+00;
      <R;
      JC    M007;
      BLD   5;
      T     LD 106;
      TAK;
      T     LD 110;
      L     P##PARAM13;
      LAR1;
      L     W [AR1,P#0.0];
      T     LW 104;
      OPN   DB [LW 104];
      L     D [AR1,P#2.0];
      LAR1;
      L     LD 110;
      L     LD 106;
      L     W [AR1,P#20.0];
M007: BLD   5;
      T     LD 106;
      TAK;
      T     LD 110;
      L     P##PARAM13;
      LAR1;
      L     W [AR1,P#0.0];
      T     LW 104;
      OPN   DB [LW 104];
      L     D [AR1,P#2.0];
      LAR1;
      L     LD 110;
      L     LD 106;
      T     W [AR1,P#20.0];
      BLD   5;
      T     LD 106;
      TAK;
      T     LD 110;
      L     P##PARAM13;
      LAR1;
      L     W [AR1,P#0.0];
      T     LW 104;
      OPN   DB [LW 104];
      L     D [AR1,P#2.0];
      LAR1;
      L     LD 110;
      L     LD 106;
      L     W [AR1,P#20.0];
      BLD   5;
      T     LD 106;
      TAK;
      T     LD 110;
      L     P##PARAM12;
      LAR1;
      L     W [AR1,P#0.0];
      T     LW 104;
      OPN   DB [LW 104];
      L     D [AR1,P#2.0];
      LAR1;
      L     LD 110;
      L     LD 106;
      T     W [AR1,P#20.0];
      BLD   5;
      T     LD 106;
      TAK;
      T     LD 110;
      L     P##PARAM12;
      LAR1;
      L     W [AR1,P#0.0];
      T     LW 104;
      OPN   DB [LW 104];
      L     D [AR1,P#2.0];
      LAR1;
      L     LD 110;
      L     LD 106;
      L     B [AR1,P#28.0];
      T     LW 30;
      L     1;
      ==I;
      JC    M008;
      L     0;
      BLD   5;
      T     LD 106;
      TAK;
      T     LD 110;
      L     P##PARAM13;
      LAR1;
      L     W [AR1,P#0.0];
      T     LW 104;
      OPN   DB [LW 104];
      L     D [AR1,P#2.0];
      LAR1;
      L     LD 110;
      L     LD 106;
      T     W [AR1,P#32.0];
      BLD   5;
      T     LD 106;
      TAK;
      T     LD 110;
      L     P##PARAM13;
      LAR1;
      L     W [AR1,P#0.0];
      T     LW 104;
      OPN   DB [LW 104];
      L     D [AR1,P#2.0];
      LAR1;
      L     LD 110;
      L     LD 106;
      T     W [AR1,P#34.0];
      BLD   5;
      T     LD 106;
      TAK;
      T     LD 110;
      L     P##PARAM13;
      LAR1;
      L     W [AR1,P#0.0];
      T     LW 104;
      OPN   DB [LW 104];
      L     D [AR1,P#2.0];
      LAR1;
      L     LD 110;
      L     LD 106;
      T     W [AR1,P#36.0];
      BLD   5;
      T     LD 106;
      TAK;
      T     LD 110;
      L     P##PARAM12;
      LAR1;
      L     W [AR1,P#0.0];
      T     LW 104;
      OPN   DB [LW 104];
      L     D [AR1,P#2.0];
      LAR1;
      L     LD 110;
      L     LD 106;
      L     B [AR1,P#28.0];
      T     LW 30;
      L     2;
      ==I;
      JC    M009;
M008: BLD   5;
      T     LD 106;
      TAK;
      T     LD 110;
      L     P##PARAM13;
      LAR1;
      L     W [AR1,P#0.0];
      T     LW 104;
      OPN   DB [LW 104];
      L     D [AR1,P#2.0];
      LAR1;
      L     LD 110;
      L     LD 106;
      L     W [AR1,P#32.0];
      BLD   5;
      T     LD 106;
      TAK;
      T     LD 110;
      L     P##PARAM12;
      LAR1;
      L     W [AR1,P#0.0];
      T     LW 104;
      OPN   DB [LW 104];
      L     D [AR1,P#2.0];
      LAR1;
      L     LD 110;
      L     LD 106;
      T     W [AR1,P#30.0];
      BLD   5;
      T     LD 106;
      TAK;
      T     LD 110;
      L     P##PARAM13;
      LAR1;
      L     W [AR1,P#0.0];
      T     LW 104;
      OPN   DB [LW 104];
      L     D [AR1,P#2.0];
      LAR1;
      L     LD 110;
      L     LD 106;
      L     W [AR1,P#34.0];
      BLD   5;
      T     LD 106;
      TAK;
      T     LD 110;
      L     P##PARAM12;
      LAR1;
      L     W [AR1,P#0.0];
      T     LW 104;
      OPN   DB [LW 104];
      L     D [AR1,P#2.0];
      LAR1;
      L     LD 110;
      L     LD 106;
      T     W [AR1,P#32.0];
      BLD   5;
      T     LD 106;
      TAK;
      T     LD 110;
      L     P##PARAM13;
      LAR1;
      L     W [AR1,P#0.0];
      T     LW 104;
      OPN   DB [LW 104];
      L     D [AR1,P#2.0];
      LAR1;
      L     LD 110;
      L     LD 106;
      L     W [AR1,P#36.0];
      BLD   5;
      T     LD 106;
      TAK;
      T     LD 110;
      L     P##PARAM12;
      LAR1;
      L     W [AR1,P#0.0];
      T     LW 104;
      OPN   DB [LW 104];
      L     D [AR1,P#2.0];
      LAR1;
      L     LD 110;
      L     LD 106;
      T     W [AR1,P#34.0];
      JU    M010;
M009: BLD   5;
      T     LD 106;
      TAK;
      T     LD 110;
      L     P##PARAM13;
      LAR1;
      L     W [AR1,P#0.0];
      T     LW 104;
      OPN   DB [LW 104];
      L     D [AR1,P#2.0];
      LAR1;
      L     LD 110;
      L     LD 106;
      L     W [AR1,P#38.0];
      BLD   5;
      T     LD 106;
      TAK;
      T     LD 110;
      L     P##PARAM12;
      LAR1;
      L     W [AR1,P#0.0];
      T     LW 104;
      OPN   DB [LW 104];
      L     D [AR1,P#2.0];
      LAR1;
      L     LD 110;
      L     LD 106;
      T     W [AR1,P#36.0];
      BLD   5;
      T     LD 106;
      TAK;
      T     LD 110;
      L     P##PARAM13;
      LAR1;
      L     W [AR1,P#0.0];
      T     LW 104;
      OPN   DB [LW 104];
      L     D [AR1,P#2.0];
      LAR1;
      L     LD 110;
      L     LD 106;
      L     W [AR1,P#40.0];
      BLD   5;
      T     LD 106;
      TAK;
      T     LD 110;
      L     P##PARAM12;
      LAR1;
      L     W [AR1,P#0.0];
      T     LW 104;
      OPN   DB [LW 104];
      L     D [AR1,P#2.0];
      LAR1;
      L     LD 110;
      L     LD 106;
      T     W [AR1,P#38.0];
      BLD   5;
      T     LD 106;
      TAK;
      T     LD 110;
      L     P##PARAM13;
      LAR1;
      L     W [AR1,P#0.0];
      T     LW 104;
      OPN   DB [LW 104];
      L     D [AR1,P#2.0];
      LAR1;
      L     LD 110;
      L     LD 106;
      L     W [AR1,P#42.0];
      BLD   5;
      T     LD 106;
      TAK;
      T     LD 110;
      L     P##PARAM12;
      LAR1;
      L     W [AR1,P#0.0];
      T     LW 104;
      OPN   DB [LW 104];
      L     D [AR1,P#2.0];
      LAR1;
      L     LD 110;
      L     LD 106;
      T     W [AR1,P#40.0];
      BLD   5;
      T     LD 106;
      TAK;
      T     LD 110;
      L     P##PARAM13;
      LAR1;
      L     W [AR1,P#0.0];
      T     LW 104;
      OPN   DB [LW 104];
      L     D [AR1,P#2.0];
      LAR1;
      L     LD 110;
      L     LD 106;
      L     W [AR1,P#44.0];
      BLD   5;
      T     LD 106;
      TAK;
      T     LD 110;
      L     P##PARAM12;
      LAR1;
      L     W [AR1,P#0.0];
      T     LW 104;
      OPN   DB [LW 104];
      L     D [AR1,P#2.0];
      LAR1;
      L     LD 110;
      L     LD 106;
      T     W [AR1,P#42.0];
      BLD   5;
      T     LD 106;
      TAK;
      T     LD 110;
      L     P##PARAM13;
      LAR1;
      L     W [AR1,P#0.0];
      T     LW 104;
      OPN   DB [LW 104];
      L     D [AR1,P#2.0];
      LAR1;
      L     LD 110;
      L     LD 106;
      L     W [AR1,P#46.0];
      BLD   5;
      T     LD 106;
      TAK;
      T     LD 110;
      L     P##PARAM12;
      LAR1;
      L     W [AR1,P#0.0];
      T     LW 104;
      OPN   DB [LW 104];
      L     D [AR1,P#2.0];
      LAR1;
      L     LD 110;
      L     LD 106;
      T     W [AR1,P#44.0];
M010: NOP   0;
NETWORK
TITLE =
// (network holds code this reader does not know; not shown)
NETWORK
TITLE =
      BLD   5;
      T     LD 106;
      TAK;
      T     LD 110;
      L     P##PARAM12;
      LAR1;
      L     W [AR1,P#0.0];
      T     LW 104;
      OPN   DB [LW 104];
      L     D [AR1,P#2.0];
      LAR1;
      L     LD 110;
      L     LD 106;
      L     W [AR1,P#20.0];
      L     LW 16;
      >=I;
      S     #PARAM8;
      BLD   5;
      T     LD 106;
      TAK;
      T     LD 110;
      L     P##PARAM12;
      LAR1;
      L     W [AR1,P#0.0];
      T     LW 104;
      OPN   DB [LW 104];
      L     D [AR1,P#2.0];
      LAR1;
      L     LD 110;
      L     LD 106;
      L     W [AR1,P#20.0];
      BLD   5;
      T     LD 106;
      TAK;
      T     LD 110;
      L     P##PARAM12;
      LAR1;
      L     W [AR1,P#0.0];
      T     LW 104;
      OPN   DB [LW 104];
      L     D [AR1,P#2.0];
      LAR1;
      L     LD 110;
      L     LD 106;
      L     W [AR1,P#18.0];
      +I;
      L     LW 16;
      <=I;
      R     #PARAM8;
      BLD   5;
      T     LD 106;
      TAK;
      T     LD 110;
      L     P##PARAM12;
      LAR1;
      L     W [AR1,P#0.0];
      T     LW 104;
      OPN   DB [LW 104];
      L     D [AR1,P#2.0];
      LAR1;
      L     LD 110;
      L     LD 106;
      L     W [AR1,P#22.0];
      L     LW 16;
      >=I;
      S     #PARAM7;
      BLD   5;
      T     LD 106;
      TAK;
      T     LD 110;
      L     P##PARAM12;
      LAR1;
      L     W [AR1,P#0.0];
      T     LW 104;
      OPN   DB [LW 104];
      L     D [AR1,P#2.0];
      LAR1;
      L     LD 110;
      L     LD 106;
      L     W [AR1,P#22.0];
      BLD   5;
      T     LD 106;
      TAK;
      T     LD 110;
      L     P##PARAM12;
      LAR1;
      L     W [AR1,P#0.0];
      T     LW 104;
      OPN   DB [LW 104];
      L     D [AR1,P#2.0];
      LAR1;
      L     LD 110;
      L     LD 106;
      L     W [AR1,P#18.0];
      +I;
      L     LW 16;
      <=I;
      R     #PARAM7;
      BLD   5;
      T     LD 106;
      TAK;
      T     LD 110;
      L     P##PARAM12;
      LAR1;
      L     W [AR1,P#0.0];
      T     LW 104;
      OPN   DB [LW 104];
      L     D [AR1,P#2.0];
      LAR1;
      L     LD 110;
      L     LD 106;
      L     W [AR1,P#24.0];
      L     LW 16;
      <=I;
      S     #PARAM6;
      BLD   5;
      T     LD 106;
      TAK;
      T     LD 110;
      L     P##PARAM12;
      LAR1;
      L     W [AR1,P#0.0];
      T     LW 104;
      OPN   DB [LW 104];
      L     D [AR1,P#2.0];
      LAR1;
      L     LD 110;
      L     LD 106;
      L     W [AR1,P#24.0];
      BLD   5;
      T     LD 106;
      TAK;
      T     LD 110;
      L     P##PARAM12;
      LAR1;
      L     W [AR1,P#0.0];
      T     LW 104;
      OPN   DB [LW 104];
      L     D [AR1,P#2.0];
      LAR1;
      L     LD 110;
      L     LD 106;
      L     W [AR1,P#18.0];
      -I;
      L     LW 16;
      >=I;
      R     #PARAM6;
      BLD   5;
      T     LD 106;
      TAK;
      T     LD 110;
      L     P##PARAM12;
      LAR1;
      L     W [AR1,P#0.0];
      T     LW 104;
      OPN   DB [LW 104];
      L     D [AR1,P#2.0];
      LAR1;
      L     LD 110;
      L     LD 106;
      L     W [AR1,P#26.0];
      L     LW 16;
      <=I;
      S     #PARAM5;
      BLD   5;
      T     LD 106;
      TAK;
      T     LD 110;
      L     P##PARAM12;
      LAR1;
      L     W [AR1,P#0.0];
      T     LW 104;
      OPN   DB [LW 104];
      L     D [AR1,P#2.0];
      LAR1;
      L     LD 110;
      L     LD 106;
      L     W [AR1,P#26.0];
      BLD   5;
      T     LD 106;
      TAK;
      T     LD 110;
      L     P##PARAM12;
      LAR1;
      L     W [AR1,P#0.0];
      T     LW 104;
      OPN   DB [LW 104];
      L     D [AR1,P#2.0];
      LAR1;
      L     LD 110;
      L     LD 106;
      L     W [AR1,P#18.0];
      -I;
      L     LW 16;
      >=I;
      R     #PARAM5;
      AN    #PARAM4;
      JC    M029;
      SET;
      =     #PARAM5;
      =     #PARAM8;
M029: NOP   0;
      BLD   5;
      T     LD 106;
      TAK;
      T     LD 110;
      L     P##PARAM12;
      LAR1;
      L     W [AR1,P#0.0];
      T     LW 104;
      OPN   DB [LW 104];
      L     D [AR1,P#2.0];
      LAR1;
      L     LD 110;
      L     LD 106;
      L     D [AR1,P#0.0];
      L     -1.000000e+02;
      <>R;
      JC    M030;
      SET;
      =     #PARAM5;
      =     #PARAM8;
M030: NOP   0;
END_FUNCTION

FUNCTION "temperature" : VOID	// FC 109
AUTHOR : gaw-be
FAMILY : temperat
NAME : display
VERSION : 0.1
BEGIN
// (block stored without names or comments; labels and parameter names are numbered)
NETWORK
TITLE =
      BLD   5;
      T     LD 10;
      TAK;
      T     LD 14;
      L     P##PARAM11;
      LAR1;
      L     W [AR1,P#0.0];
      T     LW 8;
      OPN   DB [LW 8];
      L     D [AR1,P#2.0];
      LAR1;
      L     LD 14;
      L     LD 10;
      L     W [AR1,P#34.0];
      L     -1;
      ==I;
      BLD   5;
      T     LD 10;
      TAK;
      T     LD 14;
      L     P##PARAM11;
      LAR1;
      L     W [AR1,P#0.0];
      T     LW 8;
      OPN   DB [LW 8];
      L     D [AR1,P#2.0];
      LAR1;
      L     LD 14;
      L     LD 10;
      R      [AR1,P#36.0];
      L     #PARAM2;
      BLD   5;
      T     LD 10;
      TAK;
      T     LD 14;
      L     P##PARAM11;
      LAR1;
      L     W [AR1,P#0.0];
      T     LW 8;
      OPN   DB [LW 8];
      L     D [AR1,P#2.0];
      LAR1;
      L     LD 14;
      L     LD 10;
      L     W [AR1,P#34.0];
      <>I;
      JC    M006;
      BLD   5;
      T     LD 10;
      TAK;
      T     LD 14;
      L     P##PARAM11;
      LAR1;
      L     W [AR1,P#0.0];
      T     LW 8;
      OPN   DB [LW 8];
      L     D [AR1,P#2.0];
      LAR1;
      L     LD 14;
      L     LD 10;
      A      [AR1,P#36.0];
      JC    M001;
      BLD   5;
      T     LD 10;
      TAK;
      T     LD 14;
      L     P##PARAM10;
      LAR1;
      L     W [AR1,P#0.0];
      T     LW 8;
      OPN   DB [LW 8];
      L     D [AR1,P#2.0];
      LAR1;
      L     LD 14;
      L     LD 10;
      L     B [AR1,P#4.0];
      BLD   5;
      T     LD 10;
      TAK;
      T     LD 14;
      L     P##PARAM11;
      LAR1;
      L     W [AR1,P#0.0];
      T     LW 8;
      OPN   DB [LW 8];
      L     D [AR1,P#2.0];
      LAR1;
      L     LD 14;
      L     LD 10;
      T     B [AR1,P#4.0];
      BLD   5;
      T     LD 10;
      TAK;
      T     LD 14;
      L     P##PARAM10;
      LAR1;
      L     W [AR1,P#0.0];
      T     LW 8;
      OPN   DB [LW 8];
      L     D [AR1,P#2.0];
      LAR1;
      L     LD 14;
      L     LD 10;
      L     D [AR1,P#6.0];
      BLD   5;
      T     LD 10;
      TAK;
      T     LD 14;
      L     P##PARAM11;
      LAR1;
      L     W [AR1,P#0.0];
      T     LW 8;
      OPN   DB [LW 8];
      L     D [AR1,P#2.0];
      LAR1;
      L     LD 14;
      L     LD 10;
      T     D [AR1,P#6.0];
      BLD   5;
      T     LD 10;
      TAK;
      T     LD 14;
      L     P##PARAM10;
      LAR1;
      L     W [AR1,P#0.0];
      T     LW 8;
      OPN   DB [LW 8];
      L     D [AR1,P#2.0];
      LAR1;
      L     LD 14;
      L     LD 10;
      L     D [AR1,P#10.0];
      BLD   5;
      T     LD 10;
      TAK;
      T     LD 14;
      L     P##PARAM11;
      LAR1;
      L     W [AR1,P#0.0];
      T     LW 8;
      OPN   DB [LW 8];
      L     D [AR1,P#2.0];
      LAR1;
      L     LD 14;
      L     LD 10;
      T     D [AR1,P#10.0];
      BLD   5;
      T     LD 10;
      TAK;
      T     LD 14;
      L     P##PARAM10;
      LAR1;
      L     W [AR1,P#0.0];
      T     LW 8;
      OPN   DB [LW 8];
      L     D [AR1,P#2.0];
      LAR1;
      L     LD 14;
      L     LD 10;
      L     D [AR1,P#14.0];
      BLD   5;
      T     LD 10;
      TAK;
      T     LD 14;
      L     P##PARAM11;
      LAR1;
      L     W [AR1,P#0.0];
      T     LW 8;
      OPN   DB [LW 8];
      L     D [AR1,P#2.0];
      LAR1;
      L     LD 14;
      L     LD 10;
      T     D [AR1,P#14.0];
      BLD   5;
      T     LD 10;
      TAK;
      T     LD 14;
      L     P##PARAM10;
      LAR1;
      L     W [AR1,P#0.0];
      T     LW 8;
      OPN   DB [LW 8];
      L     D [AR1,P#2.0];
      LAR1;
      L     LD 14;
      L     LD 10;
      L     D [AR1,P#18.0];
      BLD   5;
      T     LD 10;
      TAK;
      T     LD 14;
      L     P##PARAM11;
      LAR1;
      L     W [AR1,P#0.0];
      T     LW 8;
      OPN   DB [LW 8];
      L     D [AR1,P#2.0];
      LAR1;
      L     LD 14;
      L     LD 10;
      T     D [AR1,P#18.0];
      BLD   5;
      T     LD 10;
      TAK;
      T     LD 14;
      L     P##PARAM10;
      LAR1;
      L     W [AR1,P#0.0];
      T     LW 8;
      OPN   DB [LW 8];
      L     D [AR1,P#2.0];
      LAR1;
      L     LD 14;
      L     LD 10;
      L     D [AR1,P#22.0];
      BLD   5;
      T     LD 10;
      TAK;
      T     LD 14;
      L     P##PARAM11;
      LAR1;
      L     W [AR1,P#0.0];
      T     LW 8;
      OPN   DB [LW 8];
      L     D [AR1,P#2.0];
      LAR1;
      L     LD 14;
      L     LD 10;
      T     D [AR1,P#22.0];
      BLD   5;
      T     LD 10;
      TAK;
      T     LD 14;
      L     P##PARAM10;
      LAR1;
      L     W [AR1,P#0.0];
      T     LW 8;
      OPN   DB [LW 8];
      L     D [AR1,P#2.0];
      LAR1;
      L     LD 14;
      L     LD 10;
      L     D [AR1,P#26.0];
      BLD   5;
      T     LD 10;
      TAK;
      T     LD 14;
      L     P##PARAM11;
      LAR1;
      L     W [AR1,P#0.0];
      T     LW 8;
      OPN   DB [LW 8];
      L     D [AR1,P#2.0];
      LAR1;
      L     LD 14;
      L     LD 10;
      T     D [AR1,P#26.0];
      BLD   5;
      T     LD 10;
      TAK;
      T     LD 14;
      L     P##PARAM10;
      LAR1;
      L     W [AR1,P#0.0];
      T     LW 8;
      OPN   DB [LW 8];
      L     D [AR1,P#2.0];
      LAR1;
      L     LD 14;
      L     LD 10;
      L     D [AR1,P#30.0];
      BLD   5;
      T     LD 10;
      TAK;
      T     LD 14;
      L     P##PARAM11;
      LAR1;
      L     W [AR1,P#0.0];
      T     LW 8;
      OPN   DB [LW 8];
      L     D [AR1,P#2.0];
      LAR1;
      L     LD 14;
      L     LD 10;
      T     D [AR1,P#30.0];
      SET;
      BLD   5;
      T     LD 10;
      TAK;
      T     LD 14;
      L     P##PARAM11;
      LAR1;
      L     W [AR1,P#0.0];
      T     LW 8;
      OPN   DB [LW 8];
      L     D [AR1,P#2.0];
      LAR1;
      L     LD 14;
      L     LD 10;
      =      [AR1,P#36.0];
M001: BLD   5;
      T     LD 10;
      TAK;
      T     LD 14;
      L     P##PARAM10;
      LAR1;
      L     W [AR1,P#0.0];
      T     LW 8;
      OPN   DB [LW 8];
      L     D [AR1,P#2.0];
      LAR1;
      L     LD 14;
      L     LD 10;
      L     D [AR1,P#0.0];
      BLD   5;
      T     LD 10;
      TAK;
      T     LD 14;
      L     P##PARAM11;
      LAR1;
      L     W [AR1,P#0.0];
      T     LW 8;
      OPN   DB [LW 8];
      L     D [AR1,P#2.0];
      LAR1;
      L     LD 14;
      L     LD 10;
      T     D [AR1,P#0.0];
      BLD   5;
      T     LD 10;
      TAK;
      T     LD 14;
      L     P##PARAM11;
      LAR1;
      L     W [AR1,P#0.0];
      T     LW 8;
      OPN   DB [LW 8];
      L     D [AR1,P#2.0];
      LAR1;
      L     LD 14;
      L     LD 10;
      L     B [AR1,P#4.0];
      BLD   5;
      T     LD 10;
      TAK;
      T     LD 14;
      L     P##PARAM10;
      LAR1;
      L     W [AR1,P#0.0];
      T     LW 8;
      OPN   DB [LW 8];
      L     D [AR1,P#2.0];
      LAR1;
      L     LD 14;
      L     LD 10;
      T     B [AR1,P#4.0];
      BLD   5;
      T     LD 10;
      TAK;
      T     LD 14;
      L     P##PARAM11;
      LAR1;
      L     W [AR1,P#0.0];
      T     LW 8;
      OPN   DB [LW 8];
      L     D [AR1,P#2.0];
      LAR1;
      L     LD 14;
      L     LD 10;
      L     D [AR1,P#6.0];
      BLD   5;
      T     LD 10;
      TAK;
      T     LD 14;
      L     P##PARAM10;
      LAR1;
      L     W [AR1,P#0.0];
      T     LW 8;
      OPN   DB [LW 8];
      L     D [AR1,P#2.0];
      LAR1;
      L     LD 14;
      L     LD 10;
      T     D [AR1,P#6.0];
      BLD   5;
      T     LD 10;
      TAK;
      T     LD 14;
      L     P##PARAM11;
      LAR1;
      L     W [AR1,P#0.0];
      T     LW 8;
      OPN   DB [LW 8];
      L     D [AR1,P#2.0];
      LAR1;
      L     LD 14;
      L     LD 10;
      L     D [AR1,P#10.0];
      BLD   5;
      T     LD 10;
      TAK;
      T     LD 14;
      L     P##PARAM10;
      LAR1;
      L     W [AR1,P#0.0];
      T     LW 8;
      OPN   DB [LW 8];
      L     D [AR1,P#2.0];
      LAR1;
      L     LD 14;
      L     LD 10;
      T     D [AR1,P#10.0];
      BLD   5;
      T     LD 10;
      TAK;
      T     LD 14;
      L     P##PARAM11;
      LAR1;
      L     W [AR1,P#0.0];
      T     LW 8;
      OPN   DB [LW 8];
      L     D [AR1,P#2.0];
      LAR1;
      L     LD 14;
      L     LD 10;
      L     D [AR1,P#14.0];
      BLD   5;
      T     LD 10;
      TAK;
      T     LD 14;
      L     P##PARAM10;
      LAR1;
      L     W [AR1,P#0.0];
      T     LW 8;
      OPN   DB [LW 8];
      L     D [AR1,P#2.0];
      LAR1;
      L     LD 14;
      L     LD 10;
      T     D [AR1,P#14.0];
      BLD   5;
      T     LD 10;
      TAK;
      T     LD 14;
      L     P##PARAM11;
      LAR1;
      L     W [AR1,P#0.0];
      T     LW 8;
      OPN   DB [LW 8];
      L     D [AR1,P#2.0];
      LAR1;
      L     LD 14;
      L     LD 10;
      L     D [AR1,P#26.0];
      BLD   5;
      T     LD 10;
      TAK;
      T     LD 14;
      L     P##PARAM11;
      LAR1;
      L     W [AR1,P#0.0];
      T     LW 8;
      OPN   DB [LW 8];
      L     D [AR1,P#2.0];
      LAR1;
      L     LD 14;
      L     LD 10;
      L     D [AR1,P#30.0];
      >R;
      JC    M002;
      BLD   5;
      T     LD 10;
      TAK;
      T     LD 14;
      L     P##PARAM11;
      LAR1;
      L     W [AR1,P#0.0];
      T     LW 8;
      OPN   DB [LW 8];
      L     D [AR1,P#2.0];
      LAR1;
      L     LD 14;
      L     LD 10;
      L     D [AR1,P#26.0];
      BLD   5;
      T     LD 10;
      TAK;
      T     LD 14;
      L     P##PARAM11;
      LAR1;
      L     W [AR1,P#0.0];
      T     LW 8;
      OPN   DB [LW 8];
      L     D [AR1,P#2.0];
      LAR1;
      L     LD 14;
      L     LD 10;
      L     D [AR1,P#22.0];
      <R;
      JC    M002;
      BLD   5;
      T     LD 10;
      TAK;
      T     LD 14;
      L     P##PARAM11;
      LAR1;
      L     W [AR1,P#0.0];
      T     LW 8;
      OPN   DB [LW 8];
      L     D [AR1,P#2.0];
      LAR1;
      L     LD 14;
      L     LD 10;
      L     D [AR1,P#26.0];
M002: BLD   5;
      T     LD 10;
      TAK;
      T     LD 14;
      L     P##PARAM11;
      LAR1;
      L     W [AR1,P#0.0];
      T     LW 8;
      OPN   DB [LW 8];
      L     D [AR1,P#2.0];
      LAR1;
      L     LD 14;
      L     LD 10;
      T     D [AR1,P#26.0];
      BLD   5;
      T     LD 10;
      TAK;
      T     LD 14;
      L     P##PARAM11;
      LAR1;
      L     W [AR1,P#0.0];
      T     LW 8;
      OPN   DB [LW 8];
      L     D [AR1,P#2.0];
      LAR1;
      L     LD 14;
      L     LD 10;
      L     D [AR1,P#26.0];
      BLD   5;
      T     LD 10;
      TAK;
      T     LD 14;
      L     P##PARAM10;
      LAR1;
      L     W [AR1,P#0.0];
      T     LW 8;
      OPN   DB [LW 8];
      L     D [AR1,P#2.0];
      LAR1;
      L     LD 14;
      L     LD 10;
      T     D [AR1,P#26.0];
      BLD   5;
      T     LD 10;
      TAK;
      T     LD 14;
      L     P##PARAM11;
      LAR1;
      L     W [AR1,P#0.0];
      T     LW 8;
      OPN   DB [LW 8];
      L     D [AR1,P#2.0];
      LAR1;
      L     LD 14;
      L     LD 10;
      L     D [AR1,P#30.0];
      BLD   5;
      T     LD 10;
      TAK;
      T     LD 14;
      L     P##PARAM11;
      LAR1;
      L     W [AR1,P#0.0];
      T     LW 8;
      OPN   DB [LW 8];
      L     D [AR1,P#2.0];
      LAR1;
      L     LD 14;
      L     LD 10;
      L     D [AR1,P#14.0];
      >R;
      JC    M003;
      BLD   5;
      T     LD 10;
      TAK;
      T     LD 14;
      L     P##PARAM11;
      LAR1;
      L     W [AR1,P#0.0];
      T     LW 8;
      OPN   DB [LW 8];
      L     D [AR1,P#2.0];
      LAR1;
      L     LD 14;
      L     LD 10;
      L     D [AR1,P#30.0];
      BLD   5;
      T     LD 10;
      TAK;
      T     LD 14;
      L     P##PARAM11;
      LAR1;
      L     W [AR1,P#0.0];
      T     LW 8;
      OPN   DB [LW 8];
      L     D [AR1,P#2.0];
      LAR1;
      L     LD 14;
      L     LD 10;
      L     D [AR1,P#26.0];
      <R;
      JC    M003;
      BLD   5;
      T     LD 10;
      TAK;
      T     LD 14;
      L     P##PARAM11;
      LAR1;
      L     W [AR1,P#0.0];
      T     LW 8;
      OPN   DB [LW 8];
      L     D [AR1,P#2.0];
      LAR1;
      L     LD 14;
      L     LD 10;
      L     D [AR1,P#30.0];
M003: BLD   5;
      T     LD 10;
      TAK;
      T     LD 14;
      L     P##PARAM11;
      LAR1;
      L     W [AR1,P#0.0];
      T     LW 8;
      OPN   DB [LW 8];
      L     D [AR1,P#2.0];
      LAR1;
      L     LD 14;
      L     LD 10;
      T     D [AR1,P#30.0];
      BLD   5;
      T     LD 10;
      TAK;
      T     LD 14;
      L     P##PARAM11;
      LAR1;
      L     W [AR1,P#0.0];
      T     LW 8;
      OPN   DB [LW 8];
      L     D [AR1,P#2.0];
      LAR1;
      L     LD 14;
      L     LD 10;
      L     D [AR1,P#30.0];
      BLD   5;
      T     LD 10;
      TAK;
      T     LD 14;
      L     P##PARAM10;
      LAR1;
      L     W [AR1,P#0.0];
      T     LW 8;
      OPN   DB [LW 8];
      L     D [AR1,P#2.0];
      LAR1;
      L     LD 14;
      L     LD 10;
      T     D [AR1,P#30.0];
      BLD   5;
      T     LD 10;
      TAK;
      T     LD 14;
      L     P##PARAM11;
      LAR1;
      L     W [AR1,P#0.0];
      T     LW 8;
      OPN   DB [LW 8];
      L     D [AR1,P#2.0];
      LAR1;
      L     LD 14;
      L     LD 10;
      L     D [AR1,P#22.0];
      BLD   5;
      T     LD 10;
      TAK;
      T     LD 14;
      L     P##PARAM11;
      LAR1;
      L     W [AR1,P#0.0];
      T     LW 8;
      OPN   DB [LW 8];
      L     D [AR1,P#2.0];
      LAR1;
      L     LD 14;
      L     LD 10;
      L     D [AR1,P#26.0];
      >R;
      JC    M004;
      BLD   5;
      T     LD 10;
      TAK;
      T     LD 14;
      L     P##PARAM11;
      LAR1;
      L     W [AR1,P#0.0];
      T     LW 8;
      OPN   DB [LW 8];
      L     D [AR1,P#2.0];
      LAR1;
      L     LD 14;
      L     LD 10;
      L     D [AR1,P#22.0];
      BLD   5;
      T     LD 10;
      TAK;
      T     LD 14;
      L     P##PARAM11;
      LAR1;
      L     W [AR1,P#0.0];
      T     LW 8;
      OPN   DB [LW 8];
      L     D [AR1,P#2.0];
      LAR1;
      L     LD 14;
      L     LD 10;
      L     D [AR1,P#18.0];
      <R;
      JC    M004;
      BLD   5;
      T     LD 10;
      TAK;
      T     LD 14;
      L     P##PARAM11;
      LAR1;
      L     W [AR1,P#0.0];
      T     LW 8;
      OPN   DB [LW 8];
      L     D [AR1,P#2.0];
      LAR1;
      L     LD 14;
      L     LD 10;
      L     D [AR1,P#22.0];
M004: BLD   5;
      T     LD 10;
      TAK;
      T     LD 14;
      L     P##PARAM11;
      LAR1;
      L     W [AR1,P#0.0];
      T     LW 8;
      OPN   DB [LW 8];
      L     D [AR1,P#2.0];
      LAR1;
      L     LD 14;
      L     LD 10;
      T     D [AR1,P#22.0];
      BLD   5;
      T     LD 10;
      TAK;
      T     LD 14;
      L     P##PARAM11;
      LAR1;
      L     W [AR1,P#0.0];
      T     LW 8;
      OPN   DB [LW 8];
      L     D [AR1,P#2.0];
      LAR1;
      L     LD 14;
      L     LD 10;
      L     D [AR1,P#22.0];
      BLD   5;
      T     LD 10;
      TAK;
      T     LD 14;
      L     P##PARAM10;
      LAR1;
      L     W [AR1,P#0.0];
      T     LW 8;
      OPN   DB [LW 8];
      L     D [AR1,P#2.0];
      LAR1;
      L     LD 14;
      L     LD 10;
      T     D [AR1,P#22.0];
      BLD   5;
      T     LD 10;
      TAK;
      T     LD 14;
      L     P##PARAM11;
      LAR1;
      L     W [AR1,P#0.0];
      T     LW 8;
      OPN   DB [LW 8];
      L     D [AR1,P#2.0];
      LAR1;
      L     LD 14;
      L     LD 10;
      L     D [AR1,P#18.0];
      BLD   5;
      T     LD 10;
      TAK;
      T     LD 14;
      L     P##PARAM11;
      LAR1;
      L     W [AR1,P#0.0];
      T     LW 8;
      OPN   DB [LW 8];
      L     D [AR1,P#2.0];
      LAR1;
      L     LD 14;
      L     LD 10;
      L     D [AR1,P#22.0];
      >R;
      JC    M005;
      BLD   5;
      T     LD 10;
      TAK;
      T     LD 14;
      L     P##PARAM11;
      LAR1;
      L     W [AR1,P#0.0];
      T     LW 8;
      OPN   DB [LW 8];
      L     D [AR1,P#2.0];
      LAR1;
      L     LD 14;
      L     LD 10;
      L     D [AR1,P#18.0];
      BLD   5;
      T     LD 10;
      TAK;
      T     LD 14;
      L     P##PARAM11;
      LAR1;
      L     W [AR1,P#0.0];
      T     LW 8;
      OPN   DB [LW 8];
      L     D [AR1,P#2.0];
      LAR1;
      L     LD 14;
      L     LD 10;
      L     D [AR1,P#10.0];
      <R;
      JC    M005;
      BLD   5;
      T     LD 10;
      TAK;
      T     LD 14;
      L     P##PARAM11;
      LAR1;
      L     W [AR1,P#0.0];
      T     LW 8;
      OPN   DB [LW 8];
      L     D [AR1,P#2.0];
      LAR1;
      L     LD 14;
      L     LD 10;
      L     D [AR1,P#18.0];
M005: BLD   5;
      T     LD 10;
      TAK;
      T     LD 14;
      L     P##PARAM11;
      LAR1;
      L     W [AR1,P#0.0];
      T     LW 8;
      OPN   DB [LW 8];
      L     D [AR1,P#2.0];
      LAR1;
      L     LD 14;
      L     LD 10;
      T     D [AR1,P#18.0];
      BLD   5;
      T     LD 10;
      TAK;
      T     LD 14;
      L     P##PARAM11;
      LAR1;
      L     W [AR1,P#0.0];
      T     LW 8;
      OPN   DB [LW 8];
      L     D [AR1,P#2.0];
      LAR1;
      L     LD 14;
      L     LD 10;
      L     D [AR1,P#18.0];
      BLD   5;
      T     LD 10;
      TAK;
      T     LD 14;
      L     P##PARAM10;
      LAR1;
      L     W [AR1,P#0.0];
      T     LW 8;
      OPN   DB [LW 8];
      L     D [AR1,P#2.0];
      LAR1;
      L     LD 14;
      L     LD 10;
      T     D [AR1,P#18.0];
M006: NOP   0;
NETWORK
TITLE =
      L     #PARAM1;
      T     #PARAM8;
      T     LD 0;
      BLD   5;
      T     LD 10;
      TAK;
      T     LD 14;
      L     P##PARAM10;
      LAR1;
      L     W [AR1,P#0.0];
      T     LW 8;
      OPN   DB [LW 8];
      L     D [AR1,P#2.0];
      LAR1;
      L     LD 14;
      L     LD 10;
      L     D [AR1,P#14.0];
      BLD   5;
      T     LD 10;
      TAK;
      T     LD 14;
      L     P##PARAM10;
      LAR1;
      L     W [AR1,P#0.0];
      T     LW 8;
      OPN   DB [LW 8];
      L     D [AR1,P#2.0];
      LAR1;
      L     LD 14;
      L     LD 10;
      L     D [AR1,P#10.0];
      -R;
      L     LD 0;
      *R;
      L     1.000000e+02;
      /R;
      BLD   5;
      T     LD 10;
      TAK;
      T     LD 14;
      L     P##PARAM10;
      LAR1;
      L     W [AR1,P#0.0];
      T     LW 8;
      OPN   DB [LW 8];
      L     D [AR1,P#2.0];
      LAR1;
      L     LD 14;
      L     LD 10;
      L     D [AR1,P#10.0];
      +R;
      T     #PARAM9;
      T     LD 4;
      BLD   5;
      T     LD 10;
      TAK;
      T     LD 14;
      L     P##PARAM10;
      LAR1;
      L     W [AR1,P#0.0];
      T     LW 8;
      OPN   DB [LW 8];
      L     D [AR1,P#2.0];
      LAR1;
      L     LD 14;
      L     LD 10;
      L     B [AR1,P#4.0];
      L     0;
      ==I;
      JC    M007;
      BLD   5;
      T     LD 10;
      TAK;
      T     LD 14;
      L     P##PARAM10;
      LAR1;
      L     W [AR1,P#0.0];
      T     LW 8;
      OPN   DB [LW 8];
      L     D [AR1,P#2.0];
      LAR1;
      L     LD 14;
      L     LD 10;
      L     B [AR1,P#4.0];
      L     1;
      ==I;
      JC    M008;
      L     -1.000000e+02;
      JU    M009;
M007: L     LD 0;
      JU    M009;
M008: L     LD 4;
M009: BLD   5;
      T     LD 10;
      TAK;
      T     LD 14;
      L     P##PARAM10;
      LAR1;
      L     W [AR1,P#0.0];
      T     LW 8;
      OPN   DB [LW 8];
      L     D [AR1,P#2.0];
      LAR1;
      L     LD 14;
      L     LD 10;
      T     D [AR1,P#0.0];
NETWORK
TITLE =
      BLD   5;
      T     LD 10;
      TAK;
      T     LD 14;
      L     P##PARAM10;
      LAR1;
      L     W [AR1,P#0.0];
      T     LW 8;
      OPN   DB [LW 8];
      L     D [AR1,P#2.0];
      LAR1;
      L     LD 14;
      L     LD 10;
      L     D [AR1,P#18.0];
      L     LD 4;
      >=R;
      S     #PARAM7;
      BLD   5;
      T     LD 10;
      TAK;
      T     LD 14;
      L     P##PARAM10;
      LAR1;
      L     W [AR1,P#0.0];
      T     LW 8;
      OPN   DB [LW 8];
      L     D [AR1,P#2.0];
      LAR1;
      L     LD 14;
      L     LD 10;
      L     D [AR1,P#18.0];
      BLD   5;
      T     LD 10;
      TAK;
      T     LD 14;
      L     P##PARAM10;
      LAR1;
      L     W [AR1,P#0.0];
      T     LW 8;
      OPN   DB [LW 8];
      L     D [AR1,P#2.0];
      LAR1;
      L     LD 14;
      L     LD 10;
      L     D [AR1,P#6.0];
      +R;
      L     LD 4;
      <=R;
      R     #PARAM7;
      BLD   5;
      T     LD 10;
      TAK;
      T     LD 14;
      L     P##PARAM10;
      LAR1;
      L     W [AR1,P#0.0];
      T     LW 8;
      OPN   DB [LW 8];
      L     D [AR1,P#2.0];
      LAR1;
      L     LD 14;
      L     LD 10;
      L     D [AR1,P#22.0];
      L     LD 4;
      >=R;
      S     #PARAM6;
      BLD   5;
      T     LD 10;
      TAK;
      T     LD 14;
      L     P##PARAM10;
      LAR1;
      L     W [AR1,P#0.0];
      T     LW 8;
      OPN   DB [LW 8];
      L     D [AR1,P#2.0];
      LAR1;
      L     LD 14;
      L     LD 10;
      L     D [AR1,P#22.0];
      BLD   5;
      T     LD 10;
      TAK;
      T     LD 14;
      L     P##PARAM10;
      LAR1;
      L     W [AR1,P#0.0];
      T     LW 8;
      OPN   DB [LW 8];
      L     D [AR1,P#2.0];
      LAR1;
      L     LD 14;
      L     LD 10;
      L     D [AR1,P#6.0];
      +R;
      L     LD 4;
      <=R;
      R     #PARAM6;
      BLD   5;
      T     LD 10;
      TAK;
      T     LD 14;
      L     P##PARAM10;
      LAR1;
      L     W [AR1,P#0.0];
      T     LW 8;
      OPN   DB [LW 8];
      L     D [AR1,P#2.0];
      LAR1;
      L     LD 14;
      L     LD 10;
      L     D [AR1,P#26.0];
      L     LD 4;
      <=R;
      S     #PARAM5;
      BLD   5;
      T     LD 10;
      TAK;
      T     LD 14;
      L     P##PARAM10;
      LAR1;
      L     W [AR1,P#0.0];
      T     LW 8;
      OPN   DB [LW 8];
      L     D [AR1,P#2.0];
      LAR1;
      L     LD 14;
      L     LD 10;
      L     D [AR1,P#26.0];
      BLD   5;
      T     LD 10;
      TAK;
      T     LD 14;
      L     P##PARAM10;
      LAR1;
      L     W [AR1,P#0.0];
      T     LW 8;
      OPN   DB [LW 8];
      L     D [AR1,P#2.0];
      LAR1;
      L     LD 14;
      L     LD 10;
      L     D [AR1,P#6.0];
      -R;
      L     LD 4;
      >=R;
      R     #PARAM5;
      BLD   5;
      T     LD 10;
      TAK;
      T     LD 14;
      L     P##PARAM10;
      LAR1;
      L     W [AR1,P#0.0];
      T     LW 8;
      OPN   DB [LW 8];
      L     D [AR1,P#2.0];
      LAR1;
      L     LD 14;
      L     LD 10;
      L     D [AR1,P#30.0];
      L     LD 4;
      <=R;
      S     #PARAM4;
      BLD   5;
      T     LD 10;
      TAK;
      T     LD 14;
      L     P##PARAM10;
      LAR1;
      L     W [AR1,P#0.0];
      T     LW 8;
      OPN   DB [LW 8];
      L     D [AR1,P#2.0];
      LAR1;
      L     LD 14;
      L     LD 10;
      L     D [AR1,P#30.0];
      BLD   5;
      T     LD 10;
      TAK;
      T     LD 14;
      L     P##PARAM10;
      LAR1;
      L     W [AR1,P#0.0];
      T     LW 8;
      OPN   DB [LW 8];
      L     D [AR1,P#2.0];
      LAR1;
      L     LD 14;
      L     LD 10;
      L     D [AR1,P#6.0];
      -R;
      L     LD 4;
      >=R;
      R     #PARAM4;
      AN    #PARAM3;
      JC    M010;
      SET;
      =     #PARAM4;
      =     #PARAM7;
M010: NOP   0;
      BLD   5;
      T     LD 10;
      TAK;
      T     LD 14;
      L     P##PARAM10;
      LAR1;
      L     W [AR1,P#0.0];
      T     LW 8;
      OPN   DB [LW 8];
      L     D [AR1,P#2.0];
      LAR1;
      L     LD 14;
      L     LD 10;
      L     D [AR1,P#0.0];
      L     -1.000000e+02;
      <>R;
      JC    M011;
      SET;
      =     #PARAM4;
      =     #PARAM7;
M011: NOP   0;
END_FUNCTION

FUNCTION "AI_4-20" : VOID	// FC 111
AUTHOR : GAW-LK
FAMILY : ANALOG_I
NAME : BLOCK
VERSION : 0.1
BEGIN
// (block stored without names or comments; labels and parameter names are numbered)
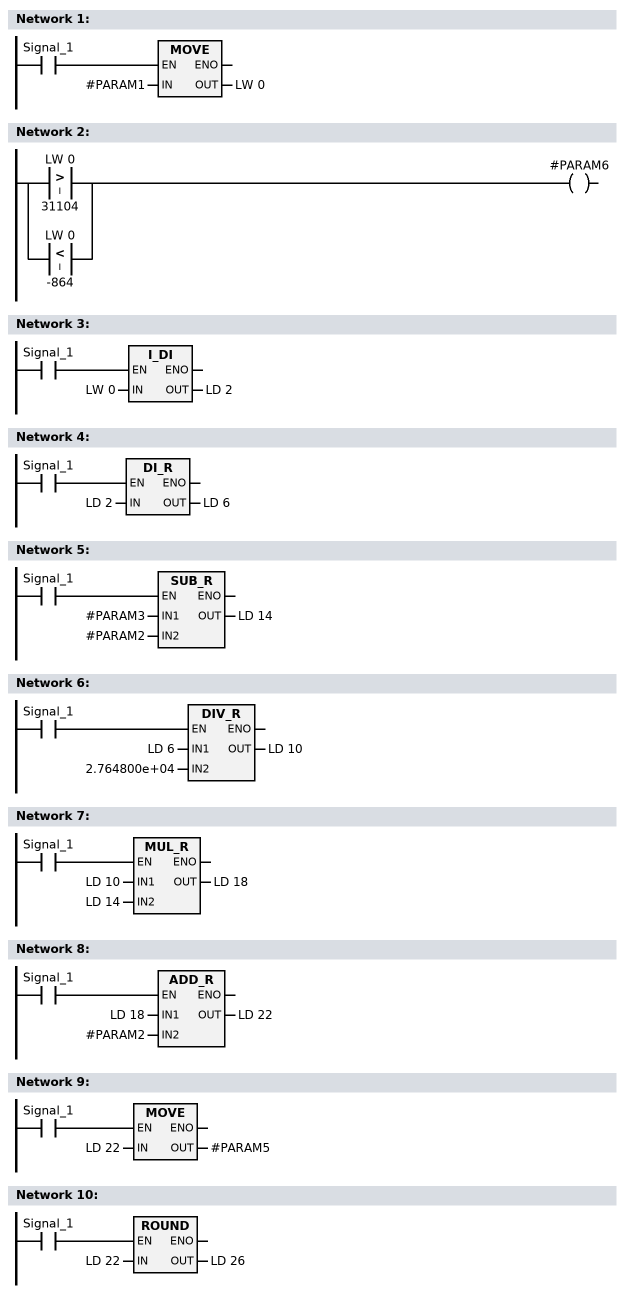
NETWORK
TITLE =
      A     "Signal_1";
      JNB   M001;
      L     #PARAM1;
      T     LW 0;
M001: NOP   0;
NETWORK
TITLE =
      O(;
      L     LW 0;
      L     31104;
      >I;
      );
      O(;
      L     LW 0;
      L     -864;
      <I;
      );
      =     #PARAM6;
NETWORK
TITLE =
      A     "Signal_1";
      JNB   M002;
      L     LW 0;
      ITD;
      T     LD 2;
M002: NOP   0;
NETWORK
TITLE =
      A     "Signal_1";
      JNB   M003;
      L     LD 2;
      DTR;
      T     LD 6;
M003: NOP   0;
NETWORK
TITLE =
      A     "Signal_1";
      JNB   M004;
      L     #PARAM3;
      L     #PARAM2;
      -R;
      T     LD 14;
M004: NOP   0;
NETWORK
TITLE =
      A     "Signal_1";
      JNB   M005;
      L     LD 6;
      L     2.764800e+04;
      /R;
      T     LD 10;
M005: NOP   0;
NETWORK
TITLE =
      A     "Signal_1";
      JNB   M006;
      L     LD 10;
      L     LD 14;
      *R;
      T     LD 18;
M006: NOP   0;
NETWORK
TITLE =
      A     "Signal_1";
      JNB   M007;
      L     LD 18;
      L     #PARAM2;
      +R;
      T     LD 22;
M007: NOP   0;
NETWORK
TITLE =
      A     "Signal_1";
      JNB   M008;
      L     LD 22;
      T     #PARAM5;
M008: NOP   0;
NETWORK
TITLE =
      A     "Signal_1";
      JNB   M009;
      L     LD 22;
      RND;
      T     LD 26;
M009: NOP   0;
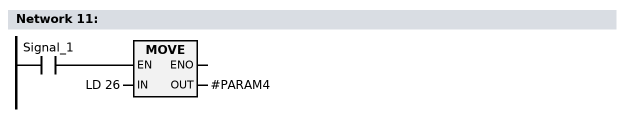
NETWORK
TITLE =
      A     "Signal_1";
      JNB   M010;
      L     LD 26;
      T     #PARAM4;
M010: NOP   0;
END_FUNCTION

